// ---- Mian/MAIN.TcPOU
// Disclaimer
// 
// This publication contains statements about the suitability of our products for certain areas of application. These statements are based on typical features of our products. The examples shown in this publication are for demonstration purposes only. 
// The information provided herein should not be regarded as specific operation characteristics. It is incumbent on the customer to check and decide whether a product is suitable for use in a particular application. 
// We do not give any warranty that the source code which is made available with this publication is complete or accurate. 
//
// THE SAMPLE CODE CONTAINED IN THIS PUBLICATION IS PROVIDED “AS IS” WITHOUT WARRANTY OF ANY KIND, EITHER EXPRESSED, IMPLIED OR STATUTORY, INCLUDING WITHOUT LIMITATION, ANY WARRANTY WITH RESPECT TO NON-INFRINGEMENT, FREEDOM FROM PROPRIETARY RIGHTS OF THIRD PARTIES OR FITNESS FOR ANY PARTICULAR PURPOSE. 
// This publication may be changed from time to time without prior notice. No liability is assumed for errors and/or omissions. Our products are described in detail in our data sheets and documentations. Product-specific warnings and cautions must be observed. 
// For the latest version of our data sheets and documentations visit our website (www.beckhoff.de). 
//
// © Beckhoff Automation GmbH & Co. KG, 2022
// The reproduction, distribution and utilization of this document as well as the communication of its contents to others without express authorization is prohibited. Offenders will be held liable for the payment of damages. All rights reserved in the event of the grant of a patent, utility model or design.
PROGRAM MAIN
VAR_INPUT
	bExecuteComplete			: BOOL;									//Command Execute Complete, not defined
END_VAR
VAR
	firstCycle : BOOL := TRUE;
	UserModeCofig				: PML_UnitModeConfig;					//User can configure his own Mode
	
	fbMachine					: FB_Machine;							//Instance of FB_Machine
//	fbMachine_2					: FB_Machine;							//Instance of FB_Machine
	bMachineStartedUp			: BOOL := FALSE;						//TRUE, when first PLC-Cycle finish
	fbVisu						: FB_Visu;								//Visualization
							//Visualization
	fbTrigger					: F_TRIG;								//Trigger for resseting Counters
	fbTrigger_2					: F_TRIG;								//Trigger for resseting Counters

	fbLocalSystemTime			 : FB_LocalSystemTime;					//Get local Systemtime
	fbLocalSystemTime_2			 : FB_LocalSystemTime;					//Get local Systemtime
	
	fbTriggerErrorMainAxis		: R_TRIG;								//Trigger for detecting Error on Mainaxis and write into PackTags
	fbTriggerErrorMetalAxis		: R_TRIG;								//Trigger for detecting Error on Metalaxis and write into PackTags
	fbTriggerErrorPlasticAxis	: R_TRIG;								//Trigger for detecting Error on Plasticaxis and write into PackTags
	
	nStateCommandCheck			: DINT;									//State to handle with statecommands
	
	i	: INT;
	tonDly	: TON;
	FB_GetUPSStatus: FB_GetUPSStatus;	
	dataloaded: BOOL;								//UPS数据文件读取状态（True为读取成功，False为读取失败）
	OldData: BOOL;									//UPS备份数据文件读取状态
	PersistentDataStatus: EPlcPersistentStatus;		//Persistent数据读取（恢复）状态	
//	fb_ups	:FB_S_UPS_CX51x0;
	//application	: FB_Application;

	bButton				: BOOL;
	ton_button			: TON;

	refMachine_control_cmd	:REFERENCE TO MachineControlCommand;
	
	refMachine_control_cmd_2	:REFERENCE TO MachineControlCommand;
	
	rTrig_error	:ARRAY[0..10] OF R_TRIG;
	rTrig_error_2	:ARRAY[0..10] OF R_TRIG;
	
	rTrig_agingTest	:R_TRIG;
	fTrig_agingTest	:F_TRIG;

	topicCallbackTest	: E_Topics;
	dataCallbackTest	: PubSubData;
	topic_sample	: E_topic_sample;
	
	(***********************ADS********************************)
	light_tower_1			:	FB_Light_tower_module;
	light_tower_2			:	FB_Light_tower_module;
   // application_1			:	FB_Application;
	tote_1					:	FB_Tote_Subsystem;
	tote_2					:	FB_Tote_Subsystem;
	safety_1				:	FB_Safety_Subsystem;
	safety_2				:	FB_Safety_Subsystem;
	machine_control_1		:	FB_MachineControl_Subsystem;
	machine_control_2		:	FB_MachineControl_Subsystem;
	heartbeat_1				:	FB_HeartBeat_Subsystem;
	heartbeat_2				:	FB_HeartBeat_Subsystem;
	
	air_pressure_1			:	FB_AirPressure_Subsystem;
	air_pressure_2			:	FB_AirPressure_Subsystem;
	
	
	heartbeat_data_test : HeartbeatParams;	
	update_light_tower_params_test	: UpdateLightTowerParams;
	tset1: UDINT;
	
	
	version 				:	STRING(255);
	testbool: BOOL;
	inbound_tote_params_test : InboundToteParams;
	OutboundToteParams_test		:	OutboundToteParams;
	testbool1: BOOL;
	
	
	
	fbMachine1					: FB_Machine;							//Instance of FB_Machine
	fbMachine2					: FB_Machine;							//Instance of FB_Machine
	stateMachine1	: FB_StateMachine;
	stateMachine2	: FB_StateMachine;
	
	
END_VAR

(**************************************UPS*****************************************)
FB_GetUPSStatus(
	sNetId:= , 					//默认为本机Netid
	nPort:= , 					//ADS端口号，若不填写功能块会自动获取，默认0
	bEnable:= , 				//高电平有效，置True后循环读取UPS状态
	bValid=> , 					//当bValid为True时，stStatus的值有效
	bError=> , 
	nErrId=> , 
	stStatus=> );				//包含UPS信息的结构体
	

dataloaded:=_Appinfo.BootDataLoaded;
OldData:=_Appinfo.OldBootData;
PersistentDataStatus:=_Appinfo.PersistentStatus;

//application();
version:='v1.0.0';

tonDly(PT:= T#10MS);
//Configure Usermode 1
A_UnitModeConfig();

//Runs the first PLC-Cycle
IF fbMachine1.bUndefinedDone AND fbMachine2.bUndefinedDone AND NOT bMachineStartedUp THEN
	GVL.PackTags1.Command.CntrlCmd	:= ePMLCommand_Abort;
	GVL.PackTags2.Command.CntrlCmd	:= ePMLCommand_Abort;
	bMachineStartedUp			:= TRUE;
END_IF


GVL.bButtonProductionReq := GVL.PackTags.Command.UnitMode = ePMLProtUnitMode_Production AND GVL.PackTags.Status.UnitModeCurrent <> GVL.PackTags.Command.UnitMode;

//Set the Packtags
M_SetPackTags();

//set the errors and warnings in Packtags
M_SetPackTagsErrorWarning();

//Call Visu
M_CallVisu();
///////////////////initialize unitmode and set 
IF GVL.PackTags.Command.UnitMode=ePMLProtUnitMode_Invalid THEN
	GVL.PackTags.Command.UnitMode	:= ePMLProtUnitMode_Production;
	GVL.PackTags.Command.Parameter[1].Value := 1;
	GVL.PackTags1.Command.UnitMode	:= ePMLProtUnitMode_Production;
	GVL.PackTags1.Command.Parameter[1].Value := 1;	
	GVL.PackTags2.Command.UnitMode	:= ePMLProtUnitMode_Production;
	GVL.PackTags2.Command.Parameter[1].Value := 1;	
	
END_IF

//Call FB_Machine
GVL.fb_working1._iModuleID:= ModuleID.WORKING1;
GVL.fb_working1._sInstanceName	:= 'working1';
GVL.fb_loading._iModuleID:= ModuleID.LOADING;
GVL.fb_loading._sInstanceName	:= 'loading';
GVL.fb_working2._iModuleID:= ModuleID.WORKING2;
GVL.fb_working2._sInstanceName	:= 'working2';
GVL.fb_loading();
GVL.fb_working1();
GVL.fb_working2();
GVL.fb_autoStore1();
GVL.fb_autoStore1._sInstanceName	:= 'autoStore_1';
GVL.fb_autoStore1._iModuleID	:= ModuleID.AUTOSTORE1;
GVL.fb_autoStore2();
GVL.fb_autoStore2._sInstanceName	:= 'autoStore_2';
GVL.fb_autoStore2._iModuleID	:= ModuleID.AUTOSTORE2;

fbMachine1(	eModeCommand:= GVL.PackTags.Command.UnitMode,
  			eMode => GVL.PackTags1.Status.UnitModeCurrent, 
			eState =>GVL.PackTags1.Status.StateCurrent,
			pPML_Instance1:=ADR(GVL.fb_working1),
			pPML_Instance2:=ADR(GVL.fb_loading),
			pPackTags:=ADR(GVL.PackTags1),
			pSafetySystem	:= ADR(safety_1)
			);
			
fbMachine2(	eModeCommand:= GVL.PackTags.Command.UnitMode,
  			eMode => GVL.PackTags2.Status.UnitModeCurrent, 
			eState =>GVL.PackTags2.Status.StateCurrent,
			pPML_Instance1:=ADR(GVL.fb_working2),
			pPML_Instance2:=ADR(GVL.fb_loading),
			pPackTags:=ADR(GVL.PackTags2),
			pSafetySystem	:= ADR(safety_2)
			);		
	
stateMachine1(	pPackTags:=ADR(GVL.PackTags1),
				pMachine:=ADR(fbMachine1),
				pMachine_control_cmd := ADR(machine_control_1.machineControlCmd),
				pAirSystem	:=ADR(air_pressure_1),
				pSafetySystem	:= ADR(safety_1),
				pMcp	:= ADR(GVL.fb_mcp_1)
				);

stateMachine2(	pPackTags:=ADR(GVL.PackTags2),
				pMachine:=ADR(fbMachine2),
				pMachine_control_cmd := ADR(machine_control_2.machineControlCmd),
				pAirSystem	:=ADR(air_pressure_2),
				pSafetySystem	:= ADR(safety_2),
				pMcp	:= ADR(GVL.fb_mcp_2)
				);			
		
			
GVL.fbWriteLog(
	bWrite:= GVL.bWrite, 
	sFileName:= , 
	sMessage:= , 
	OK=> , 
	Busy=> , 
	ErrorMsg=> , 
	bError=> , 
	ErrorID=> );
	
(***********************ADS********************************)
GVL.fb_mcp_1(id:=1);
GVL.fb_mcp_2(id:=2);
tote_1();
safety_1(pHeartBeat:=ADR(heartbeat_1),pSafety_door:=ADR(GVL.fb_mcp_1.st_safety_door),pPackTags:=ADR(GVL.PackTags1),pMachine:=ADR(fbMachine1));
air_pressure_1(pPackTags:=ADR(GVL.PackTags1));
heartbeat_1();
light_tower_1(pHeartBeat:=ADR(heartbeat_1),pLightTower:= ADR(GVL.fb_mcp_1.lightTower));
machine_control_1(pMachineCurrentStatus:= ADR(GVL.PackTags1.Status.StateCurrent));
tote_1._sInstanceName	:='tote_1';
safety_1._sInstanceName	:='safety_1';
air_pressure_1._sInstanceName	:='air_pressure1';

tote_2();
light_tower_2(pHeartBeat:=ADR(heartbeat_2),pLightTower:= ADR(GVL.fb_mcp_2.lightTower));
safety_2(pHeartBeat:=ADR(heartbeat_2),pSafety_door:=ADR(GVL.fb_mcp_2.st_safety_door),pPackTags:=ADR(GVL.PackTags2),pMachine:=ADR(fbMachine2));
air_pressure_2(pPackTags:=ADR(GVL.PackTags2));
heartbeat_2();
machine_control_2(pMachineCurrentStatus:= ADR(GVL.PackTags2.Status.StateCurrent));
tote_2._sInstanceName	:='tote_2';
safety_2._sInstanceName	:='safety_2';
air_pressure_2._sInstanceName	:='air_pressure2';


M_SetUnitInfo();

ACTION A_UnitModeConfig:
UserModeCofig(
	eMode							:= ePMLUnitMode_Service, 
	bDisableClearing				:= TRUE, 
	bDisableStarting				:= FALSE, 
	bDisableSuspended				:= FALSE, 
	bDisableStopping				:= TRUE, 
	bDisableAborting				:= TRUE, 
	bDisableHolding					:= TRUE, 
	bDisableHeld					:= TRUE, 
	bDisableUnholding				:= TRUE, 
	bDisableSuspending				:= TRUE, 
	bDisableUnsuspending			:= TRUE, 
	bDisableResetting				:= TRUE, 
	bDisableIdle					:= FALSE, 
	bDisableCompleting				:= TRUE, 
	bDisableComplete				:= FALSE, 
	bEnableUnitModeChangeStopped	:= TRUE, 
	bEnableUnitModeChangeIdle		:= TRUE, 
	bEnableUnitModeChangeSuspended	:= FALSE, 
	bEnableUnitModeChangeExecute	:= FALSE, 
	bEnableUnitModeChangeAborted	:= TRUE, 
	bEnableUnitModeChangeHeld		:= FALSE, 
	bEnableUnitModeChangeComplete	:= TRUE, 
	bError							=> , 
	nErrorId						=> );
UserModeCofig(
	eMode							:= ePMLUnitMode_Production, 
	bDisableClearing				:= FALSE, 
	bDisableStarting				:= FALSE, 
	bDisableSuspended				:= TRUE, 
	bDisableStopping				:= FALSE, 
	bDisableAborting				:= FALSE, 
	bDisableHolding					:= TRUE, 
	bDisableHeld					:= TRUE, 
	bDisableUnholding				:= TRUE, 
	bDisableSuspending				:= TRUE, 
	bDisableUnsuspending			:= TRUE, 
	bDisableResetting				:= FALSE, 
	bDisableIdle					:= FALSE, 
	bDisableCompleting				:= FALSE, 
	bDisableComplete				:= FALSE, 
	bEnableUnitModeChangeStopped	:= TRUE, 
	bEnableUnitModeChangeIdle		:= TRUE, 
	bEnableUnitModeChangeSuspended	:= FALSE, 
	bEnableUnitModeChangeExecute	:= FALSE, 
	bEnableUnitModeChangeAborted	:= TRUE, 
	bEnableUnitModeChangeHeld		:= FALSE, 
	bEnableUnitModeChangeComplete	:= TRUE, 
	bError							=> , 
	nErrorId						=> );
END_ACTION

METHOD M_CallVisu
VAR_INPUT
END_VAR
//Calling FB_Visu
fbVisu(
	aKeyPressed				:= GVL.aKeyPressed,
	aUnitInfo				:= GVL.aUnitInfo, 
	bInvalidEntry			=> ,
	aCaption				=> GVL.aCaption,
	eModeVisu				=> ,
	eStateVisu				=> ,
	sUnitName				=> ,
	iFrameVisible			=> );
END_METHOD

METHOD M_SetPackTags
VAR_INPUT
END_VAR
VAR	
END_VAR
//***************************Writing Data into GVL.PackTags***************************

//Parameters for the production
GVL.PackTags.Command.Parameter[1].ID				:= 1;
GVL.PackTags.Command.Parameter[1].Name				:= 'Quantity';
GVL.PackTags.Command.Parameter[1].Unit				:= 'Tote';

//Countig produced totes, see fb_sample1
GVL.PackTags.Admin.ProdProcessedCount[1].ID			:= 1;
GVL.PackTags.Admin.ProdProcessedCount[1].Name		:= 'ToteFinish_Sample';
GVL.PackTags.Admin.ProdProcessedCount[1].Unit		:= 'Tote';





//Write the actual state and mode into the GVL.PackTags
GVL.PackTags.Status.StateCurrent					:= fbMachine1.eState;
GVL.PackTags.Status.UnitModeCurrent					:= fbMachine1.eMode;
GVL.PackTags.Status.StateRequested					:= fbMachine1.eCommand;
GVL.PackTags.Status.UnitModeRequested				:= fbMachine1.eModeCommand;
GVL.PackTags.Status.StateChangeInProcess			:= GVL.PackTags.Status.StateCurrent <> GVL.PackTags.Status.StateRequested;
GVL.PackTags.Status.UnitModeChangeInProcess			:= GVL.PackTags.Status.UnitModeCurrent <> GVL.PackTags.Status.UnitModeRequested;

//Write the actual state and mode into the GVL.PackTags2
GVL.PackTags1.Status.StateCurrent					:= fbMachine1.eState;
GVL.PackTags1.Status.UnitModeCurrent					:= fbMachine1.eMode;
GVL.PackTags1.Status.StateRequested					:= fbMachine1.eCommand;
GVL.PackTags1.Status.UnitModeRequested				:= fbMachine1.eModeCommand;
GVL.PackTags1.Status.StateChangeInProcess			:= GVL.PackTags1.Status.StateCurrent <> GVL.PackTags1.Status.StateRequested;
GVL.PackTags1.Status.UnitModeChangeInProcess			:= GVL.PackTags1.Status.UnitModeCurrent <> GVL.PackTags1.Status.UnitModeRequested;
//Write the actual state and mode into the GVL.PackTags2
GVL.PackTags2.Status.StateCurrent					:= fbMachine2.eState;
GVL.PackTags2.Status.UnitModeCurrent					:= fbMachine2.eMode;
GVL.PackTags2.Status.StateRequested					:= fbMachine2.eCommand;
GVL.PackTags2.Status.UnitModeRequested				:= fbMachine2.eModeCommand;
GVL.PackTags2.Status.StateChangeInProcess			:= GVL.PackTags2.Status.StateCurrent <> GVL.PackTags2.Status.StateRequested;
GVL.PackTags2.Status.UnitModeChangeInProcess			:= GVL.PackTags2.Status.UnitModeCurrent <> GVL.PackTags2.Status.UnitModeRequested;


//Write actual time and date in GVL.PackTags
fbLocalSystemTime(sNetID:= '', bEnable := TRUE);
GVL.PackTags.Admin.PlcDateTime[0]	:= fbLocalSystemTime.systemTime.wYear;
GVL.PackTags.Admin.PlcDateTime[1]	:= fbLocalSystemTime.systemTime.wMonth;
GVL.PackTags.Admin.PlcDateTime[2]	:= fbLocalSystemTime.systemTime.wDay;
GVL.PackTags.Admin.PlcDateTime[3]	:= fbLocalSystemTime.systemTime.wHour;
GVL.PackTags.Admin.PlcDateTime[4]	:= fbLocalSystemTime.systemTime.wMinute;
GVL.PackTags.Admin.PlcDateTime[5]	:= fbLocalSystemTime.systemTime.wSecond;
GVL.PackTags.Admin.PlcDateTime[6]	:= fbLocalSystemTime.systemTime.wMilliseconds;
GVL.PackTags1.Admin.PlcDateTime	:= GVL.PackTags.Admin.PlcDateTime;
GVL.PackTags2.Admin.PlcDateTime	:= GVL.PackTags.Admin.PlcDateTime;
//Set the productcounter to 0, when the production command is completed
fbTrigger(CLK:= (fbMachine1.eState = ePMLState_Complete));
IF fbTrigger.Q OR GVL.stChangeIntoProduction.bYesReset THEN
	GVL.PackTags1.Admin.ProdProcessedCount[1].Count	:= 0;
	GVL.PackTags1.Command.Parameter[1].Value			:= 0;
	GVL.nVisuProductCommand							:= 0;
END_IF

//Set the productcounter to 0, when the production command is completed
fbTrigger(CLK:= (fbMachine2.eState = ePMLState_Complete));
IF fbTrigger.Q OR GVL.stChangeIntoProduction.bYesReset THEN
	GVL.PackTags2.Admin.ProdProcessedCount[1].Count	:= 0;
	GVL.PackTags2.Command.Parameter[1].Value			:= 0;
	GVL.nVisuProductCommand							:= 0;
END_IF
END_METHOD

METHOD M_SetPackTagsErrorWarning
VAR_INPUT
END_VAR
//====================Error and Warnig setting========================
//Warnings
GVL.PackTags1.Admin.Warning[1].Message	:= 'Invalid Production Command, command Products must be higher than 0';
GVL.PackTags1.Admin.Warning[1].ID 		:= 1;

GVL.PackTags1.Admin.Warning[2].Message	:= 'Invalid Mode Command, please try anothereone';
GVL.PackTags1.Admin.Warning[2].ID		:= 2;


//====================Error and Warnig handling========================
//warning for invalid production command
IF 	GVL.PackTags1.Status.UnitModeCurrent = ePMLProtUnitMode_Production AND 
	GVL.PackTags1.Status.StateCurrent = ePMLState_Idle AND 
	GVL.PackTags1.Command.CntrlCmd = ePMLCommand_Start AND
 	GVL.PackTags1.Command.Parameter[1].Value <= 0 
THEN
	GVL.PackTags1.Admin.Warning[1].Trigger :=TRUE;
ELSE
	GVL.PackTags1.Admin.Warning[1].Trigger :=FALSE;
END_IF

//warning for invalid mode command
IF fbMachine1.bInvalidModeCommandOut THEN
	GVL.PackTags1.Admin.Warning[2].Trigger :=TRUE;
ELSE 
	GVL.PackTags1.Admin.Warning[2].Trigger :=FALSE;
END_IF





//====================Error and Warnig setting========================
//Warnings
GVL.PackTags1.Admin.Warning[1].Message	:= 'Invalid Production Command, command Products must be higher than 0';
GVL.PackTags1.Admin.Warning[1].ID 		:= 1;

GVL.PackTags1.Admin.Warning[2].Message	:= 'Invalid Mode Command, please try anothereone';
GVL.PackTags1.Admin.Warning[2].ID		:= 2;


//====================Error and Warnig handling========================
//warning for invalid production command
IF 	GVL.PackTags2.Status.UnitModeCurrent = ePMLProtUnitMode_Production AND 
	GVL.PackTags2.Status.StateCurrent = ePMLState_Idle AND 
	GVL.PackTags2.Command.CntrlCmd = ePMLCommand_Start AND
 	GVL.PackTags2.Command.Parameter[1].Value <= 0 
THEN
	GVL.PackTags2.Admin.Warning[1].Trigger :=TRUE;
ELSE
	GVL.PackTags2.Admin.Warning[1].Trigger :=FALSE;
END_IF

//warning for invalid mode command
IF fbMachine2.bInvalidModeCommandOut THEN
	GVL.PackTags2.Admin.Warning[2].Trigger :=TRUE;
ELSE 
	GVL.PackTags2.Admin.Warning[2].Trigger :=FALSE;
END_IF
END_METHOD

METHOD M_SetUnitInfo
VAR_INPUT
END_VAR
GVL.aUnitInfo[eMachine1].Name			:= 'fbMachine1';
GVL.aUnitInfo[eMachine1].ActMode			:= fbMachine1.eMode;
GVL.aUnitInfo[eMachine1].ActState		:= fbMachine1.eState;

GVL.aUnitInfo[eMachine1].Name			:= 'fbMachine2';
GVL.aUnitInfo[eMachine1].ActMode		:= fbMachine2.eMode;
GVL.aUnitInfo[eMachine1].ActState		:= fbMachine2.eState;

//GVL.aUnitInfo[eSample].Name				:= GVL.fb_sample._sInstanceName;
//GVL.aUnitInfo[eSample].ActMode			:= GVL.fb_sample.eMode;
//GVL.aUnitInfo[eSample].ActState			:= GVL.fb_sample.eState;


GVL.aUnitInfo[eLoading].Name			:= GVL.fb_loading._sInstanceName;
GVL.aUnitInfo[eLoading].ActMode			:= GVL.fb_loading.eMode;
GVL.aUnitInfo[eLoading].ActState		:= GVL.fb_loading.eState;


GVL.aUnitInfo[eWorking1].Name			:= GVL.fb_working1._sInstanceName;
GVL.aUnitInfo[eWorking1].ActMode		:= GVL.fb_working1.eMode;
GVL.aUnitInfo[eWorking1].ActState		:= GVL.fb_working1.eState;


GVL.aUnitInfo[eWorking2].Name			:= GVL.fb_working2._sInstanceName;
GVL.aUnitInfo[eWorking2].ActMode		:= GVL.fb_working2.eMode;
GVL.aUnitInfo[eWorking2].ActState		:= GVL.fb_working2.eState;
END_METHOD

END_PROGRAM

// ---- Mian/FB_StateMachine.TcPOU
FUNCTION_BLOCK FB_StateMachine
VAR_INPUT
	
	pPackTags				: POINTER TO ST_PackMLv30;
	pMachine				: POINTER TO FB_Machine;	
	pMachine_control_cmd	: POINTER TO MachineCommandStructure;	
	pAirSystem				: POINTER TO FB_AirPressure_Subsystem;
	pSafetySystem			: POINTER TO FB_Safety_Subsystem;	
	pMcp					: POINTER TO FB_mcp;
END_VAR
VAR_OUTPUT
END_VAR
VAR
	rTrig_error	:ARRAY[1..10] OF R_TRIG;
	i	: INT;
		

END_VAR

(*command from 1:PLC HMI buttons;2:APP;3:Safety module;4:each modules*)
/////////////////////////////abort/////////////////////////////	
IF 	pMachine^.eState <> ePMLState_Aborted AND pMachine^.eState <> ePMLState_Clearing THEN	
	IF pPackTags^.Command.CntrlCmd = ePMLCommand_Abort OR M_CheckError() THEN
		IF pMachine^.M_UnitsActive(ePMLCommand_Abort) THEN
			pMachine^.eCommand	:= ePMLCommand_Abort;
			pMachine_control_cmd^.command	:= MachineControlCommand.DO_NOTHING;
		END_IF
	END_IF
END_IF
/////////////////////////////stop/////////////////////////////
IF M_CheckError() THEN
	//
ELSE					
	IF (pPackTags^.Command.CntrlCmd = ePMLCommand_Stop OR 
		pMachine_control_cmd^.command = MachineControlCommand.STOP OR 
		pSafetySystem^.pml_command=ePMLCommand_Stop) AND pMachine^.eState <> ePMLState_Stopped
	THEN
		IF pMachine^.M_UnitsActive(ePMLCommand_Stop) THEN
			pMachine^.eCommand	:= ePMLCommand_Stop;
		END_IF
	END_IF
END_IF

CASE pMachine^.eState OF
			
	ePMLState_Aborted:
		IF pMcp^.st_safety_door.button_reset THEN
			pPackTags^.Command.CntrlCmd := ePMLCommand_Clear;
		END_IF
		IF 	pPackTags^.Command.CntrlCmd = ePMLCommand_Clear OR
			(pSafetySystem^.safety_status=SafetyStatus.READY AND pMachine_control_cmd^.command=MachineControlCommand.RESET)//while safety is ready,can be reset remotely	 
		THEN
			IF pSafetySystem^.M_reset() THEN	//reset safety first
				IF pSafetySystem^.xError THEN
					pPackTags^.Command.CntrlCmd		:= ePMLCommand_Undefined;
					pMachine_control_cmd^.command	:= MachineControlCommand.DO_NOTHING;
				ELSE
					IF pMachine^.M_UnitsActive(ePMLCommand_Clear) THEN
						pMachine^.eCommand	:= ePMLCommand_Clear;
					END_IF					
				END_IF
			END_IF	
		END_IF
		//reset command
		IF pMachine^.eCommand = ePMLCommand_Abort THEN
			pMachine^.eCommand	:= ePMLCommand_Undefined;
		END_IF
			
	ePMLState_Complete:		
		IF (pPackTags^.Command.CntrlCmd = ePMLCommand_Reset OR pMachine_control_cmd^.command = MachineControlCommand.RESET (*OR
		 	pMcp^.st_safety_door.button_reset*)) 
		THEN
			pMachine^.eCommand	:= ePMLCommand_Reset;
		END_IF
			
			
	ePMLState_Idle:
		IF (pPackTags^.Command.CntrlCmd = ePMLCommand_Start OR pMachine_control_cmd^.command = MachineControlCommand.START)	AND
			(NOT (pPackTags^.Command.Parameter[1].Value <= 0) OR NOT (pMachine^.eMode = 1))
		THEN	
			IF pMachine^.M_UnitsActive(ePMLCommand_Start) THEN
				pMachine^.eCommand	:= ePMLCommand_Start;
			END_IF
		END_IF
		IF pMachine_control_cmd^.command = MachineControlCommand.RESET THEN
			pMachine_control_cmd^.command	:= MachineControlCommand.DO_NOTHING;
		END_IF
		//reset command
		IF pMachine^.eCommand = ePMLCommand_Reset THEN
			pMachine^.eCommand	:= ePMLCommand_Undefined;
		END_IF
			
			
	ePMLState_Stopped:
		IF pPackTags^.Command.CntrlCmd = ePMLCommand_Reset OR pMachine_control_cmd^.command = MachineControlCommand.RESET THEN		
			IF pMachine^.M_UnitsActive(ePMLCommand_Reset) THEN
				pMachine^.eCommand	:= ePMLCommand_Reset;
			END_IF
		END_IF		
		IF (pPackTags^.Command.CntrlCmd = ePMLCommand_Start OR pMachine_control_cmd^.command = MachineControlCommand.START)	AND
			(NOT (pPackTags^.Command.Parameter[1].Value <= 0) OR NOT (pMachine^.eMode = 1)) AND
			stPMLUnitModeConfiguration[pMachine^.eMode].aStateDisabled[ePMLState_Idle] 
		THEN	
			IF pMachine^.M_UnitsActive(ePMLCommand_Start) THEN
				pMachine^.eCommand	:= ePMLCommand_Start; 	
			END_IF			
		END_IF	
		IF pMachine_control_cmd^.command = MachineControlCommand.STOP THEN
			pMachine_control_cmd^.command	:= MachineControlCommand.DO_NOTHING;
		END_IF	
		//reset command
		IF pMachine^.eCommand = ePMLCommand_Clear OR pMachine^.eCommand = ePMLCommand_Stop THEN
			pMachine^.eCommand	:= ePMLCommand_Undefined;
		END_IF
			
			
	ePMLState_Execute:	
		IF pMachine_control_cmd^.command = MachineControlCommand.START THEN
			pMachine_control_cmd^.command	:= MachineControlCommand.DO_NOTHING;
		END_IF
		IF pPackTags^.Command.CntrlCmd = ePMLCommand_Hold	AND	
			(pMachine^.eMode =  1 OR pMachine^.eMode =  4 OR pMachine^.eMode = 2)  
		THEN
			pMachine^.eCommand	:= ePMLCommand_Hold;
		END_IF	
		IF pPackTags^.Command.CntrlCmd = ePMLCommand_Suspend AND (pMachine^.eMode = 4 OR pMachine^.eMode = 1)THEN
		 
			pMachine^.eCommand	:= ePMLCommand_Suspend;
		END_IF	 
		//reset command
		IF pMachine^.eCommand = ePMLCommand_Start THEN
			pMachine^.eCommand	:= ePMLCommand_Undefined;
		END_IF
			
			
	ePMLState_Held:	 
		IF pPackTags^.Command.CntrlCmd = ePMLCommand_Unhold THEN
			pMachine^.eCommand	:= ePMLCommand_Unhold;
		END_IF
			
			
	ePMLState_Suspended:
		IF pPackTags^.Command.CntrlCmd = ePMLCommand_Unsuspend THEN
			pMachine^.eCommand	:= ePMLCommand_Unsuspend;
		END_IF
			
			
	ePMLState_Aborting,ePMLState_Clearing,ePMLState_Resetting,ePMLState_Starting,ePMLState_Stopping:
		pPackTags^.Command.CntrlCmd	:= ePMLCommand_Undefined;

		
		
END_CASE

METHOD M_CheckError : BOOL

VAR
	
END_VAR
M_CheckError	:= FALSE;

FOR i:=1 TO GlobalParameters.MaxAlarms DO
	IF pPackTags^.Admin.Alarm[i].Trigger THEN
		M_CheckError	:= TRUE;
	END_IF
END_FOR
//RETURN;//remove this while safety and air is ready
IF pSafetySystem^.xError OR pAirSystem^.air_pressure_status=AirPressureStatus.ERROR THEN
	M_CheckError	:= TRUE;
END_IF
END_METHOD

END_FUNCTION_BLOCK

// ---- GlobalTextList.TcGTLO
TEXTLIST GlobalTextList
  1242 = '    UNKNOWN := 0 \n   VACANT :=  1\n      LOADED := 2\n AWAITING_INBOUND_AVAILABILITY := 3 \n      INBOUNDING := 4\n  AWAITING_OUTBOUND_AVAILABILITY:5\n    OUTBOUNDING := 6\n    PERTURBING := 7\n    UNKNOWN_ERROR := 50, \n    MECHANICAL_ERROR := 51,\n    ELECTRICAL_ERROR := 52,\n    SAFETY_ERROR := 53,\n    UPSTREAM_NOT_READY := 54,\n    TIMEOUT_WAITING_FOR_NEW_TOTE := 55,\n    DOWNSTREAM_NOT_READY := 56,\n    TIMEOUT_WAITING_FOR_SPACE := 57,\n\tBAG_OPEN_FAILED := 100'
  1602 = '    UNKNOWN := 0 \n   VACANT :=  1\n      LOADED := 2\n AWAITING_INBOUND_AVAILABILITY := 3, \n      INBOUNDING := 4,\n  AWAITING_OUTBOUND_AVAILABILITY:5, \n    OUTBOUNDING := 6,  \n    PERTURBING := 7, \n    UNKNOWN_ERROR := 50, \n    MECHANICAL_ERROR := 51,\n    ELECTRICAL_ERROR := 52,\n    SAFETY_ERROR := 53,\n    UPSTREAM_NOT_READY := 54,\n    TIMEOUT_WAITING_FOR_NEW_TOTE := 55,\n    DOWNSTREAM_NOT_READY := 56,\n    TIMEOUT_WAITING_FOR_SPACE := 57,\n\tBAG_OPEN_FAILED := 100'
  133 = '    UNKNOWN := 0 \n   VACANT :=  1\n      LOADED := 2 AWAITING_INBOUND_AVAILABILITY := 3, \n      INBOUNDING := 4,  AWAITING_OUTBOUND_AVAILABILITY:5, \n    OUTBOUNDING := 6,  \n    PERTURBING := 7, \n    UNKNOWN_ERROR := 50, \n    MECHANICAL_ERROR := 51,\n    ELECTRICAL_ERROR := 52,\n    SAFETY_ERROR := 53,\n    UPSTREAM_NOT_READY := 54,\n    TIMEOUT_WAITING_FOR_NEW_TOTE := 55,\n    DOWNSTREAM_NOT_READY := 56,\n    TIMEOUT_WAITING_FOR_SPACE := 57,\n\tBAG_OPEN_FAILED := 100'
  1738 = '    UNKNOWN := 0 \n   VACANT :=  1，\n      LOADED := 2，\n AWAITING_INBOUND_AVAILABILITY := 3, \n      INBOUNDING := 4,\n  AWAITING_OUTBOUND_AVAILABILITY:5, \n    OUTBOUNDING := 6,  \n    PERTURBING := 7, \n    UNKNOWN_ERROR := 50, \n    MECHANICAL_ERROR := 51,\n    ELECTRICAL_ERROR := 52,\n    SAFETY_ERROR := 53,\n    UPSTREAM_NOT_READY := 54,\n    TIMEOUT_WAITING_FOR_NEW_TOTE := 55,\n    DOWNSTREAM_NOT_READY := 56,\n    TIMEOUT_WAITING_FOR_SPACE := 57,\n\tBAG_OPEN_FAILED := 100'
  3042 = '    UNKNOWN := 0 \n   VACANT :=  1，\n      LOADED := 2，\n AWAITING_INBOUND_AVAILABILITY := 3, \n      INBOUNDING := 4,  AWAITING_OUTBOUND_AVAILABILITY:5, \n    OUTBOUNDING := 6,  \n    PERTURBING := 7, \n    UNKNOWN_ERROR := 50, \n    MECHANICAL_ERROR := 51,\n    ELECTRICAL_ERROR := 52,\n    SAFETY_ERROR := 53,\n    UPSTREAM_NOT_READY := 54,\n    TIMEOUT_WAITING_FOR_NEW_TOTE := 55,\n    DOWNSTREAM_NOT_READY := 56,\n    TIMEOUT_WAITING_FOR_SPACE := 57,\n\tBAG_OPEN_FAILED := 100'
  298 = '    UNKNOWN := 0 \n   VACANT :=  1，\n      LOADED := 2， AWAITING_INBOUND_AVAILABILITY := 3, \n      INBOUNDING := 4,  AWAITING_OUTBOUND_AVAILABILITY:5, \n    OUTBOUNDING := 6,  \n    PERTURBING := 7, \n    UNKNOWN_ERROR := 50, \n    MECHANICAL_ERROR := 51,\n    ELECTRICAL_ERROR := 52,\n    SAFETY_ERROR := 53,\n    UPSTREAM_NOT_READY := 54,\n    TIMEOUT_WAITING_FOR_NEW_TOTE := 55,\n    DOWNSTREAM_NOT_READY := 56,\n    TIMEOUT_WAITING_FOR_SPACE := 57,\n\tBAG_OPEN_FAILED := 100'
  387 = '    UNKNOWN := 0, \n    VACANT := 1\n    LOADED := 2,  AWAITING_INBOUND_AVAILABILITY := 3,  \n     INBOUNDING := 4,      AWAITING_OUTBOUND_AVAILABILITY := 5,  \n    OUTBOUNDING := 6,\n    PERTURBING := 7, \n    UNKNOWN_ERROR := 50, \n    MECHANICAL_ERROR := 51,\n    ELECTRICAL_ERROR := 52,\n    SAFETY_ERROR := 53,\n    UPSTREAM_NOT_READY := 54,\n    TIMEOUT_WAITING_FOR_NEW_TOTE := 55,\n    DOWNSTREAM_NOT_READY := 56,\n    TIMEOUT_WAITING_FOR_SPACE := 57,\n\t\n\tBAG_OPEN_FAILED := 100'
  1866 = '    UNKNOWN := 0, \n   VACANT :=  1,  \n      LOADED :=  2,  AWAITING_INBOUND_AVAILABILITY := 3, \n      INBOUNDING := 4,  AWAITING_OUTBOUND_AVAILABILITY:5, \n    OUTBOUNDING := 6,  \n    PERTURBING := 7, \n    UNKNOWN_ERROR := 50, \n    MECHANICAL_ERROR := 51,\n    ELECTRICAL_ERROR := 52,\n    SAFETY_ERROR := 53,\n    UPSTREAM_NOT_READY := 54,\n    TIMEOUT_WAITING_FOR_NEW_TOTE := 55,\n    DOWNSTREAM_NOT_READY := 56,\n    TIMEOUT_WAITING_FOR_SPACE := 57,\n\tBAG_OPEN_FAILED := 100'
  2213 = '    UNKNOWN := 0, \n   VACANT := 1,  \n    LOADED := 2,  AWAITING_INBOUND_AVAILABILITY := 3, \n      INBOUNDING := 4,  AWAITING_OUTBOUND_AVAILABILITY:5, \n    OUTBOUNDING := 6,  \n    PERTURBING := 7, \n    UNKNOWN_ERROR := 50, \n    MECHANICAL_ERROR := 51,\n    ELECTRICAL_ERROR := 52,\n    SAFETY_ERROR := 53,\n    UPSTREAM_NOT_READY := 54,\n    TIMEOUT_WAITING_FOR_NEW_TOTE := 55,\n    DOWNSTREAM_NOT_READY := 56,\n    TIMEOUT_WAITING_FOR_SPACE := 57,\n\tBAG_OPEN_FAILED := 100'
  972 = '    UNKNOWN := 0, \n   VACANT := 1,  \n    LOADED := 2,  AWAITING_INBOUND_AVAILABILITY := 3,  \n      INBOUNDING := 4,  AWAITING_OUTBOUND_AVAILABILITY := 5,  \n    OUTBOUNDING := 6,  \n    PERTURBING := 7, \n    UNKNOWN_ERROR := 50, \n    MECHANICAL_ERROR := 51,\n    ELECTRICAL_ERROR := 52,\n    SAFETY_ERROR := 53,\n    UPSTREAM_NOT_READY := 54,\n    TIMEOUT_WAITING_FOR_NEW_TOTE := 55,\n    DOWNSTREAM_NOT_READY := 56,\n    TIMEOUT_WAITING_FOR_SPACE := 57,\n\t\n\tBAG_OPEN_FAILED := 100'
  599 = '    UNKNOWN := 0, \n   VACANT := 1,  \n    LOADED := 2,  AWAITING_INBOUND_AVAILABILITY := 3,  \n      INBOUNDING := 4,  AWAITING_OUTBOUND_AVAILABILITY := 5,  \n    OUTBOUNDING := 6,  \n    PERTURBING := 7, \n    UNKNOWN_ERROR := 50, \n    MECHANICAL_ERROR := 51,\n    ELECTRICAL_ERROR := 52,\n    SAFETY_ERROR := 53,\n    UPSTREAM_NOT_READY := 54,\n    TIMEOUT_WAITING_FOR_NEW_TOTE := 55,\n    DOWNSTREAM_NOT_READY := 56,\n    TIMEOUT_WAITING_FOR_SPACE := 57,\n\tBAG_OPEN_FAILED := 100'
  2173 = '    UNKNOWN := 0,  (* when system is down *)\n    VACANT := 1, (* no tote here *)\n    LOADED := 2,  (* a tote loaded in current position *)\n    AWAITING_INBOUND_AVAILABILITY := 3,  (* waiting for an available inbound tote *)\n    INBOUNDING := 4,  (* inbounding tote from upper line *)\n    AWAITING_OUTBOUND_AVAILABILITY := 5,  (* waiting for an available outbound space *)\n    OUTBOUNDING := 6,  (* outbound tote to lower line *)\n    PERTURBING := 7, (* Tote vibrating *)\n\n    UNKNOWN_ERROR := 50, (* in error state, we should extend the error in the future\t*)\n    MECHANICAL_ERROR := 51,\n    ELECTRICAL_ERROR := 52,\n    SAFETY_ERROR := 53,\n    UPSTREAM_NOT_READY := 54,\n    TIMEOUT_WAITING_FOR_NEW_TOTE := 55,\n    DOWNSTREAM_NOT_READY := 56,\n    TIMEOUT_WAITING_FOR_SPACE := 57,\n\t\n\tBAG_OPEN_FAILED := 100'
  55 = ' command Products: %i'
  323 = '%.2f'
  206 = '%.2f mm'
  829 = '%.2f MPa'
  1131 = '%.2r'
  740 = '%.3f mm'
  201 = '%s'
  209 = '+'
  210 = '-'
  2384 = '2 Systems'
  54 = 'A C C I D E N T'
  18 = 'Abort'
  394 = 'ABORT INBOUND'
  2668 = 'ABORT OUTBOUND'
  33 = 'Aborted'
  34 = 'Aborting'
  602 = 'Acc'
  843 = 'Actual Position'
  830 = 'Admin'
  773 = 'Aging test'
  5 = 'Alarm'
  61 = 'Average MachSpeed: %5.2f Package/min'
  203 = 'Axis Error '
  299 = 'Axis_bagOpen_0'
  618 = 'Axis_bagOpen_1'
  211 = 'Axis_bagOpen_2'
  743 = 'Axis_bagOpen_3'
  324 = 'Axis_vacuun_0'
  786 = 'Axis_vacuun_1'
  317 = 'BAFFLE SENSOR1'
  1963 = 'BAFFLE SENSOR2'
  179 = 'BagOpen'
  63 = 'BagOpening'
  11 = 'BagOpening '
  521 = 'BagOpening-1'
  1064 = 'BagOpening_1'
  2321 = 'BagOpening_2'
  2069 = 'BagOpening_Detection'
  959 = 'Bag_)'
  1353 = 'Bag_0'
  1316 = 'Bag_1'
  1317 = 'Bag_closed'
  517 = 'Bag_opened'
  1009 = 'Bag_preopen'
  2196 = 'bDisplay'
  81 = 'BELT ESTOP'
  1803 = 'bLoad_up'
  808 = 'Breaker OFF'
  486 = 'Breaker ON'
  2216 = 'Btton Start'
  1159 = 'buffer'
  327 = 'BUFFER SAFETY'
  732 = 'Buffer Stopper'
  481 = 'bUsingOpenBag'
  1712 = 'Button stop'
  1438 = 'b_EStopRestart'
  16 = 'Clear'
  32 = 'Clearing'
  17 = 'Command'
  38 = 'Complete'
  1085 = 'Completing'
  58 = 'CurrentMachSpeed:%5.2f Package/min'
  1975 = 'DateTime'
  1723 = 'Datetime'
  349 = 'Dec'
  216 = 'deg/s'
  217 = 'deg/s²'
  50 = 'Detection\nof metal'
  180 = 'DIO'
  68 = 'Do you want to change tp production mode?'
  662 = 'DOG'
  2636 = 'DOOR CLOSED'
  2225 = 'Door Closed'
  1080 = 'Down'
  673 = 'error'
  586 = 'EStop Restart'
  2274 = 'EStopRestart'
  23 = 'Execute'
  19 = 'Execute\nComplete'
  924 = 'Extend'
  2482 = 'extend'
  614 = 'extended'
  59 = 'Finished Metalboxes: %i'
  60 = 'Finished Plasticboxes: %i'
  56 = 'Finished Products: %i '
  801 = 'Flood Light'
  1197 = 'GVL_IOLink'
  25 = 'Held'
  12 = 'Hold'
  26 = 'Holding'
  841 = 'HOME'
  248 = 'HomeDone'
  902 = 'ID'
  21 = 'Idle'
  136 = 'inbound'
  134 = 'INBOUND'
  710 = 'inbound_1'
  1624 = 'inbound_2'
  44 = 'INIT'
  4 = 'Invalid'
  1037 = 'Lamp'
  2490 = 'LIFT DOOR LEFT'
  2284 = 'LIFT DOOR RIGHT'
  668 = 'LIFT STO EDM'
  473 = 'Lift_down'
  293 = 'Lift_iuo'
  316 = 'Lift_up'
  51 = 'Light\nsensor'
  2749 = 'LIGHT STO EDM'
  319 = 'Load'
  1648 = 'Load Tote'
  1129 = 'Load Tote Request'
  762 = 'Loading'
  416 = 'Load_up'
  581 = 'Lock MCP Left Door'
  222 = 'Lock MCP Right Door'
  580 = 'Log In'
  234 = 'Log Out'
  1496 = 'LogOut'
  6 = 'Mantainance'
  7 = 'Manual'
  2290 = 'MCP ESTOP LEFT'
  1000 = 'MCP ESTOP RIGHT'
  1593 = 'MCP ESTOP2'
  708 = 'Message'
  361 = 'Method'
  2239 = 'MID SAFETY DOOR1'
  2485 = 'MID SAFETY DOOR2'
  52 = 'Move belt\n+'
  53 = 'Move to\nwork position'
  491 = 'Muanal'
  737 = 'name'
  3 = 'No'
  1516 = 'NO.'
  258 = 'NO. '
  1043 = 'None'
  1736 = 'Open MCP Left Door'
  1323 = 'Open MCP Right Door'
  711 = 'Operator'
  1406 = 'OUTBOUND'
  381 = 'outbound_1'
  1368 = 'outbound_2'
  1318 = 'outbound_assist\n\n'
  760 = 'outbound_assist_1\n\n'
  182 = 'outbound_assist_2\n\n'
  1029 = 'outbound_end'
  787 = 'Pause'
  1446 = 'photosensor'
  2037 = 'photo_sensor_bottom'
  1081 = 'photo_sensor_diagonal'
  706 = 'photo_sens[1]or_start'
  1231 = 'PICKMODULE STO EDM'
  882 = 'PICKMODULE2 STO EDM'
  1922 = 'PLACE1 STO EDM'
  1263 = 'PLACE2 STO EDM'
  1450 = 'PML '
  598 = 'Position Setting'
  1051 = 'Production'
  57 = 'Reset the Visu'
  30 = 'Reseting'
  176 = 'ROBO2T ESTOP'
  40 = 'ROBOT1 EAS'
  1399 = 'ROBOT1 EES'
  2581 = 'ROBOT1 ESTOP'
  1167 = 'ROBOT2 EAS'
  2067 = 'ROBOT2 EES'
  1126 = 'ROLLER BELT STO EDM'
  1023 = 'rolleroutbound_assist\n\n'
  1305 = 'roller_assign'
  1160 = 'roller_inbound'
  1610 = 'roller_inbound_assist'
  2157 = 'roller_outbound'
  1295 = 'roller_outbound_assist\n\n'
  2362 = 'SAFETY DOOR LEFT'
  1331 = 'SAFETYDOOR RIGHT'
  1925 = 'Sample'
  36 = 'SC'
  1012 = 'sensor[0]'
  1257 = 'sensor[1]'
  82 = 'sensor[2]'
  774 = 'sensor[3]'
  1262 = 'sensor[4]'
  1137 = 'sensor[5]'
  794 = 'sensor[6]'
  512 = 'sensor[7]'
  2929 = 'sensor_lift_atDownPos'
  681 = 'sensor_start[0]'
  1006 = 'sensor_start[1]'
  2179 = 'sensor_transfer_atFeedingPos'
  3056 = 'sensor_transfer_atWorkingPos'
  62 = 'Seperated Boxes: %i'
  415 = 'Service'
  102 = 'sStepID'
  99 = 'Jerk'
  839 = 'JOG BW'
  840 = 'JOG FW'
  1374 = 'lift'
  795 = 'LIFT'
  178 = 'Lift'
  926 = 'LIFT ESTOP'
  519 = 'LIFT STATION DETECTION'
  495 = 'LIGHT CURTAIN LEFT'
  39 = 'LIGHT CURTAIN RIGHT'
  413 = 'LOAD'
  897 = 'LOADING SAFETY'
  351 = 'Main'
  386 = 'MCP ESTOP'
  215 = 'mm/s'
  214 = 'mm/s²'
  207 = 'MOVE ABS'
  569 = 'Move relative'
  205 = 'Neg LS'
  677 = 'outbound'
  842 = 'photosensor[0]'
  79 = 'photosensor[1]'
  70 = 'photo_sensor[0]'
  919 = 'photo_sensor[1]'
  800 = 'photo_sensor_mute'
  925 = 'photo_sensor_mute_l'
  891 = 'photo_sensor_start'
  1003 = 'place'
  204 = 'Pos LS'
  844 = 'Power \nOn'
  359 = 'Power On'
  342 = 'ReM'
  1185 = 'ReM3'
  904 = 'ReM4'
  274 = 'ReM5'
  199 = 'Reset'
  10 = 'RESET'
  1651 = 'retract'
  934 = 'retracted'
  71 = 'ROBOT EAS'
  312 = 'ROBOT EES'
  72 = 'roller'
  1437 = 'Roller In'
  189 = 'roller[0]'
  709 = 'roller[1]'
  633 = 'roller[2]'
  687 = 'roller[3]'
  522 = 'roller_x'
  792 = 'roller_y'
  845 = 'RUN'
  634 = 'SAFETY DOOR'
  202 = 'SAFETY INPUT'
  617 = 'SAFETY OUTPUT'
  641 = 'sComponentID'
  438 = 'sComponent_ID'
  358 = 'sComponent_name'
  874 = 'sensor_mute'
  143 = 'sensor_mute_left'
  487 = 'sensor_mute_right'
  622 = 'Set absolute\nencoder as linear'
  454 = 'Set absolute\nencoder as rotation'
  208 = 'Set Point'
  14 = 'Set Pos to 0'
  332 = 'sEventType'
  714 = 'sEvent_MSG'
  245 = 'sID'
  220 = 'sMethod'
  1077 = 'Start'
  22 = 'Starting'
  67 = 'State Model\n%s'
  1356 = 'Station1'
  1785 = 'Station2'
  1034 = 'StepID'
  986 = 'sTime'
  198 = 'Stop'
  996 = 'STOP'
  1671 = 'stop'
  31 = 'Stopped'
  35 = 'Stopping'
  1097 = 'Suspend'
  28 = 'Suspended'
  29 = 'Suspending'
  666 = 'Time'
  2038 = 'time_detection'
  2651 = 'Tote1'
  1283 = 'Tote2'
  784 = 'tote_detection'
  1613 = 'TryRunMode'
  590 = 'TryRunStart'
  118 = 'TryRunStop'
  585 = 'Type'
  13 = 'Unhold'
  24 = 'Unholding'
  20 = 'Unit Mode'
  780 = 'UNLOAD'
  809 = 'Unload'
  2590 = 'Unload To Left'
  297 = 'Unload To Right'
  37 = 'Unsuspend'
  27 = 'Unsuspending'
  15 = 'Unuspend'
  407 = 'UP'
  505 = 'Up'
  848 = 'User'
  8 = 'UserMode 1'
  863 = 'valve_clamp[0]'
  1846 = 'valve_left_door'
  1781 = 'valve_left_door extend'
  2324 = 'valve_left_door valve_left_door.extend'
  676 = 'valve_left_door.extend'
  1741 = 'valve_lif'
  396 = 'valve_lift'
  464 = 'valve_lift[0]'
  247 = 'valve_lift_1'
  1409 = 'valve_lift_2'
  2061 = 'valve_lif_1'
  1819 = 'valve_right_door'
  227 = 'valve_stopper'
  200 = 'Velocity'
  193 = 'WORKING SAFETY'
  246 = 'Working1'
  753 = 'Working1 Load'
  928 = 'Working1 Unload'
  514 = 'Working2'
  2337 = 'Working2 Load'
  86 = 'Working2 Unload'
  1 = 'Yes'
  2 = 'Yes, with Reset'
END_TEXTLIST

// ---- VISUs/Templates/visu_autoStore.TcVIS
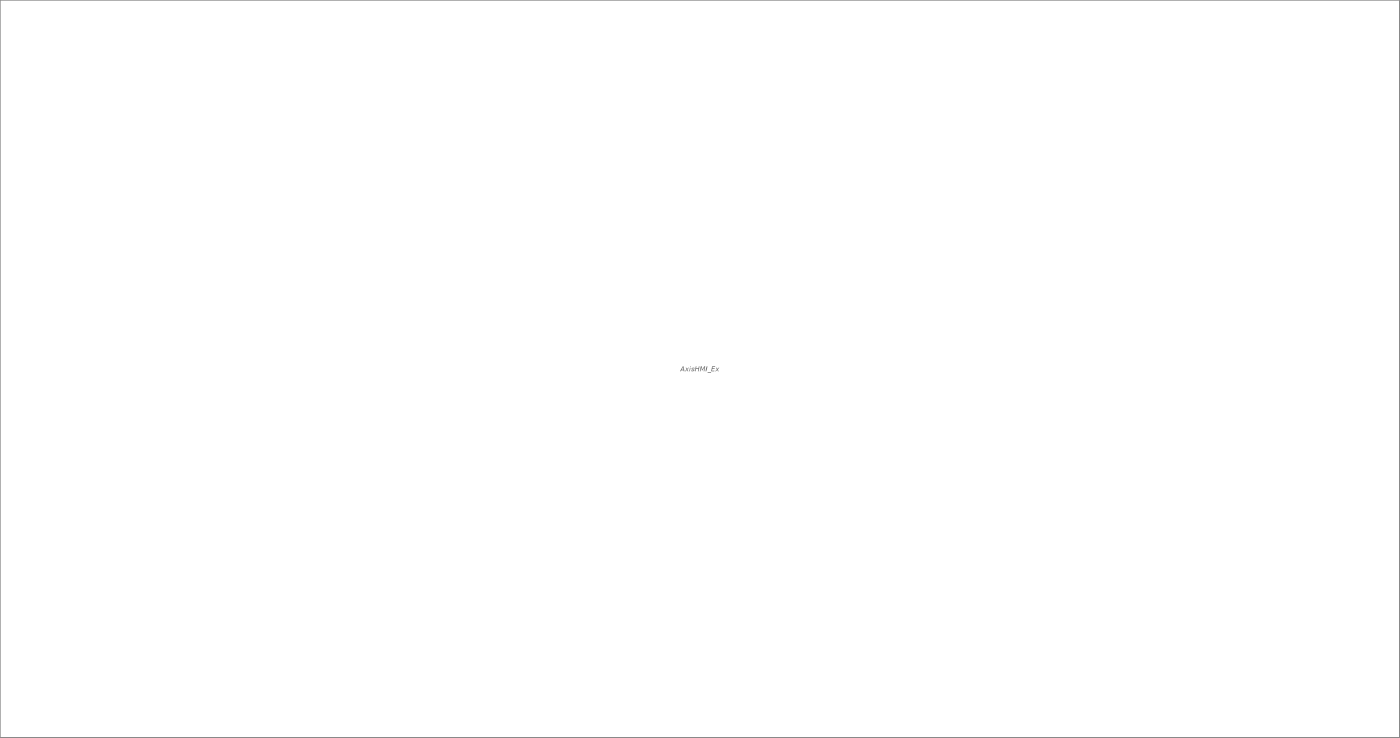
VISUALIZATION visu_autoStore  // 2048x1080
VAR_IN_OUT
	autoStore	: FB_autoStore;
END_VAR
    TabControl (0,0 2048x1080)
        shows AxisHMI_Ex(stAxisHMI := autoStore.st_mcAxis_lift, mcAxis := autoStore.mcAxis_lift, xError := autoStore.mcAxis_lift.xError)
        shows AxisHMI_Ex(stAxisHMI := autoStore.st_mcAxis_transfer, mcAxis := autoStore.mcAxis_transfer, xError := autoStore.mcAxis_transfer.xError)
        shows v_io_autoStore(autoStore := autoStore)
        shows AxisHMI_Ex(stAxisHMI := GVL.fb_working.st_mcAxis_vacuun[0], mcAxis := GVL.fb_working.mcAxis_vacuun[0], xError := GVL.fb_working.mcAxis_vacuun[0].xError)
        shows AxisHMI_Ex(stAxisHMI := GVL.fb_working.st_mcAxis_vacuun[1], mcAxis := GVL.fb_working.mcAxis_vacuun[1], xError := GVL.fb_working.mcAxis_vacuun[1].xError)
        shows AxisHMI_Ex(stAxisHMI := GVL.fb_working.st_mcAxis_bagOpen[0], mcAxis := GVL.fb_working.mcAxis_bagOpen[0], xError := GVL.fb_working.mcAxis_bagOpen[0].xError)
        shows AxisHMI_Ex(stAxisHMI := GVL.fb_working.st_mcAxis_bagOpen[1], mcAxis := GVL.fb_working.mcAxis_bagOpen[1], xError := GVL.fb_working.mcAxis_bagOpen[1].xError)
        shows AxisHMI_Ex(stAxisHMI := GVL.fb_working.st_mcAxis_bagOpen[2], mcAxis := GVL.fb_working.mcAxis_bagOpen[2], xError := GVL.fb_working.mcAxis_bagOpen[2].xError)
        shows AxisHMI_Ex(stAxisHMI := GVL.fb_working.st_mcAxis_bagOpen[3], mcAxis := GVL.fb_working.mcAxis_bagOpen[3], xError := GVL.fb_working.mcAxis_bagOpen[3].xError)
        [0]: TabTitle=Lift
        [1]: TabTitle=BagOpen
        [3]: TabTitle=Axis_vacuun_0
        [4]: TabTitle=Axis_vacuun_1
        [5]: TabTitle=Axis_bagOpen_0
        [6]: TabTitle=Axis_bagOpen_1
        [7]: TabTitle=Axis_bagOpen_2
        [8]: TabTitle=Axis_bagOpen_3
        p2837713833: gantrybase.mcAxis[EN_Axis.Z].sAxisName
END_VISUALIZATION

// ---- VISUs/Templates/VIS_TemplatePMLStateModel.TcVIS
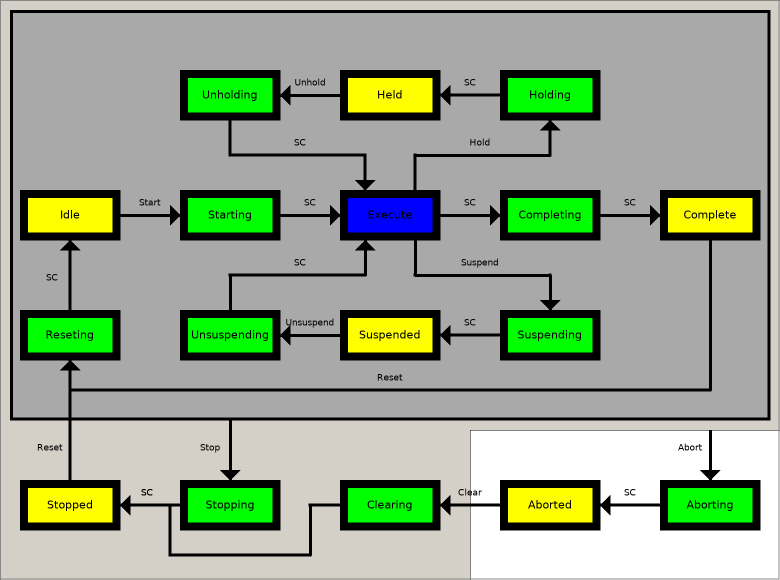
VISUALIZATION VIS_TemplatePMLStateModel  // 780x580
VAR_INPUT
	ePMLUnitMode		: DINT;
	ePMLState			: DINT;
END_VAR
VAR_IN_OUT
	eStateCommand		: DINT;
END_VAR
    Polygon (0,0) (780,0) (780,430) (470,430) (470,580) (0,580)
    Rectangle (10,10 760x410)
    Polyline (415,190) (415,155) (550,155) (550,95) (440,95), invisible if: stPMLUnitModeConfiguration[ePMLUnitMode].aStateDisabled[11]
    Polyline (365,190) (365,155) (230,155) (230,95) (340,95), invisible if: stPMLUnitModeConfiguration[ePMLUnitMode].aStateDisabled[11]
    Polyline (415,240) (415,275) (550,275) (550,335) (440,335), invisible if: stPMLUnitModeConfiguration[ePMLUnitMode].aStateDisabled[5]
    Polyline (365,240) (365,275) (230,275) (230,335) (340,335), invisible if: stPMLUnitModeConfiguration[ePMLUnitMode].aStateDisabled[5]
    Polyline (710,430) (710,505) (310,505) (310,555) (170,555) (170,505) (70,505) (70,215) (340,215)
    RoundedRectangle (20,190 100x50), "Idle", colour toggle: (ePMLState = 4), invisible if: stPMLUnitModeConfiguration[ePMLUnitMode].aStateDisabled[4]
    RoundedRectangle (180,190 100x50), "Starting", colour toggle: (ePMLState = 3), invisible if: stPMLUnitModeConfiguration[ePMLUnitMode].aStateDisabled[3]
    RoundedRectangle (340,190 100x50), "Execute", colour toggle: (ePMLState = 6)
    RoundedRectangle (180,70 100x50), "Unholding", colour toggle: (ePMLState = 12), invisible if: stPMLUnitModeConfiguration[ePMLUnitMode].aStateDisabled[12]
    RoundedRectangle (340,70 100x50), "Held", colour toggle: (ePMLState = 11), invisible if: stPMLUnitModeConfiguration[ePMLUnitMode].aStateDisabled[11]
    RoundedRectangle (500,70 100x50), "Holding", colour toggle: (ePMLState = 10), invisible if: stPMLUnitModeConfiguration[ePMLUnitMode].aStateDisabled[10]
    RoundedRectangle (180,310 100x50), "Unsuspending", colour toggle: (ePMLState = 14), invisible if: stPMLUnitModeConfiguration[ePMLUnitMode].aStateDisabled[14]
    RoundedRectangle (340,310 100x50), "Suspended", colour toggle: (ePMLState = 5), invisible if: stPMLUnitModeConfiguration[ePMLUnitMode].aStateDisabled[5]
    RoundedRectangle (500,310 100x50), "Suspending", colour toggle: (ePMLState = 13), invisible if: stPMLUnitModeConfiguration[ePMLUnitMode].aStateDisabled[13]
    RoundedRectangle (20,310 100x50), "Reseting", colour toggle: (ePMLState = 15), invisible if: stPMLUnitModeConfiguration[ePMLUnitMode].aStateDisabled[15]
    RoundedRectangle (20,480 100x50), "Stopped", colour toggle: (ePMLState = 2)
    RoundedRectangle (340,480 100x50), "Clearing", colour toggle: (ePMLState = 1), invisible if: stPMLUnitModeConfiguration[ePMLUnitMode].aStateDisabled[1]
    RoundedRectangle (500,480 100x50), "Aborted", colour toggle: (ePMLState = 9)
    RoundedRectangle (660,480 100x50), "Aborting", colour toggle: (ePMLState = 8), invisible if: stPMLUnitModeConfiguration[ePMLUnitMode].aStateDisabled[8]
    Polygon (550,120) (540,130) (560,130), invisible if: stPMLUnitModeConfiguration[ePMLUnitMode].aStateDisabled[10]
    Polygon (365,240) (355,250) (375,250), invisible if: stPMLUnitModeConfiguration[ePMLUnitMode].aStateDisabled[5]
    Polygon (70,240) (60,250) (80,250), invisible if: stPMLUnitModeConfiguration[ePMLUnitMode].aStateDisabled[4]
    Polygon (70,360) (60,370) (80,370), invisible if: stPMLUnitModeConfiguration[ePMLUnitMode].aStateDisabled[15]
    Polygon (440,95) (450,105) (450,85), invisible if: stPMLUnitModeConfiguration[ePMLUnitMode].aStateDisabled[11]
    Polygon (280,95) (290,105) (290,85), invisible if: stPMLUnitModeConfiguration[ePMLUnitMode].aStateDisabled[12]
    Polygon (440,335) (450,345) (450,325), invisible if: stPMLUnitModeConfiguration[ePMLUnitMode].aStateDisabled[5]
    Polygon (280,335) (290,345) (290,325), invisible if: stPMLUnitModeConfiguration[ePMLUnitMode].aStateDisabled[14]
    Polygon (600,505) (610,515) (610,495)
    Polygon (440,505) (450,515) (450,495), invisible if: stPMLUnitModeConfiguration[ePMLUnitMode].aStateDisabled[1]
    Polygon (120,505) (130,515) (130,495)
    Polygon (180,215) (170,225) (170,205), invisible if: stPMLUnitModeConfiguration[ePMLUnitMode].aStateDisabled[3]
    Polygon (340,215) (330,225) (330,205)
    Polygon (500,215) (490,225) (490,205), invisible if: stPMLUnitModeConfiguration[ePMLUnitMode].aStateDisabled[16]
    Polygon (660,215) (650,225) (650,205), invisible if: stPMLUnitModeConfiguration[ePMLUnitMode].aStateDisabled[17]
    Polygon (375,180) (365,190) (355,180), invisible if: stPMLUnitModeConfiguration[ePMLUnitMode].aStateDisabled[11]
    Polygon (560,300) (550,310) (540,300), invisible if: stPMLUnitModeConfiguration[ePMLUnitMode].aStateDisabled[13]
    Polygon (720,470) (710,480) (700,470), invisible if: stPMLUnitModeConfiguration[ePMLUnitMode].aStateDisabled[8]
    Polygon (240,470) (230,480) (220,470), invisible if: stPMLUnitModeConfiguration[ePMLUnitMode].aStateDisabled[7]
    Polyline (230,420) (230,505) (150,505)
    RoundedRectangle (180,480 100x50), "Stopping", colour toggle: (ePMLState = 7), invisible if: stPMLUnitModeConfiguration[ePMLUnitMode].aStateDisabled[7]
    Label (440,135 80x15), "Hold", invisible if: stPMLUnitModeConfiguration[ePMLUnitMode].aStateDisabled[11]
    Label (260,135 80x15), "SC", invisible if: stPMLUnitModeConfiguration[ePMLUnitMode].aStateDisabled[12]
    Label (430,75 80x15), "SC", invisible if: stPMLUnitModeConfiguration[ePMLUnitMode].aStateDisabled[10]
    Label (270,75 80x15), "Unhold", invisible if: stPMLUnitModeConfiguration[ePMLUnitMode].aStateDisabled[11]
    Label (270,315 80x15), "Unsuspend", invisible if: stPMLUnitModeConfiguration[ePMLUnitMode].aStateDisabled[5]
    Label (430,315 80x15), "SC", invisible if: stPMLUnitModeConfiguration[ePMLUnitMode].aStateDisabled[13]
    Label (440,255 80x15), "Suspend", invisible if: stPMLUnitModeConfiguration[ePMLUnitMode].aStateDisabled[5]
    Label (260,255 80x15), "SC", invisible if: stPMLUnitModeConfiguration[ePMLUnitMode].aStateDisabled[14]
    Label (270,195 80x15), "SC", invisible if: stPMLUnitModeConfiguration[ePMLUnitMode].aStateDisabled[3]
    Label (590,195 80x15), "SC", invisible if: stPMLUnitModeConfiguration[ePMLUnitMode].aStateDisabled[16]
    Label (430,195 80x15), "SC", invisible if: stPMLUnitModeConfiguration[ePMLUnitMode].aStateDisabled[17]
    Label (430,485 80x15), "Clear"
    Label (590,485 80x15), "SC", invisible if: stPMLUnitModeConfiguration[ePMLUnitMode].aStateDisabled[8]
    Label (107,485 80x15), "SC", invisible if: stPMLUnitModeConfiguration[ePMLUnitMode].aStateDisabled[1]
    Label (350,370 80x15), "Reset", invisible if: stPMLUnitModeConfiguration[ePMLUnitMode].aStateDisabled[17]
    Label (10,440 80x15), "Reset", invisible if: stPMLUnitModeConfiguration[ePMLUnitMode].aStateDisabled[4]
    Label (170,440 80x15), "Stop"
    Label (650,440 80x15), "Abort"
    Label (12,270 80x15), "SC", invisible if: stPMLUnitModeConfiguration[ePMLUnitMode].aStateDisabled[15]
    Label (110,195 80x15), "Start"
    Label (107,485 80x15), "SC", invisible if: stPMLUnitModeConfiguration[ePMLUnitMode].aStateDisabled[7]
    Polyline (440,215) (710,215) (710,390) (70,390), invisible if: stPMLUnitModeConfiguration[ePMLUnitMode].aStateDisabled[17]
    RoundedRectangle (660,190 100x50), "Complete", colour toggle: (ePMLState = 17), invisible if: stPMLUnitModeConfiguration[ePMLUnitMode].aStateDisabled[17]
    RoundedRectangle (500,190 100x50), "Completing", colour toggle: (ePMLState = 16), invisible if: stPMLUnitModeConfiguration[ePMLUnitMode].aStateDisabled[16]
END_VISUALIZATION

// ---- VISUs/Templates/v_io_autoStore.TcVIS
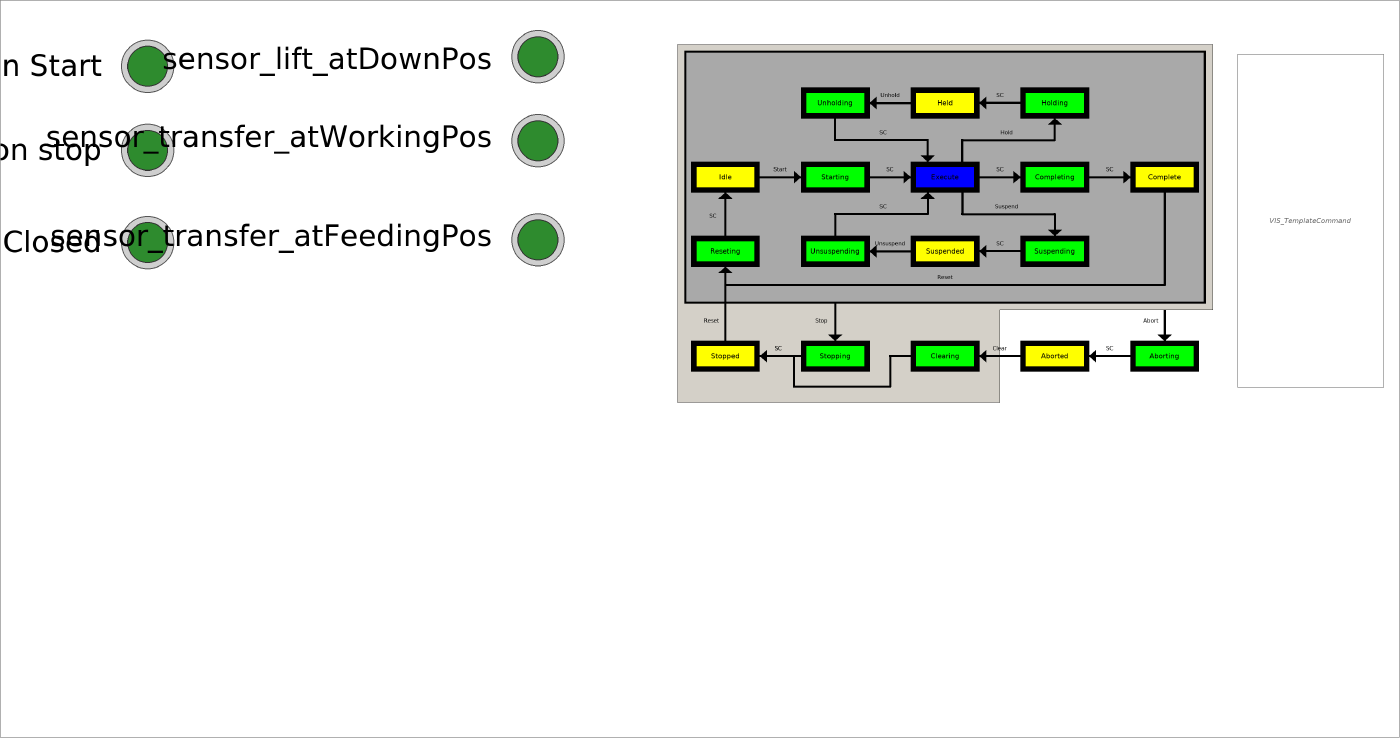
VISUALIZATION v_io_autoStore  // 2048x1080
VAR_IN_OUT
	autoStore	: FB_autoStore;
END_VAR
    Lamp1 (171,52 90x90), variable: autoStore.button_start, style: Lamp-Lamp1-Green
    Label (32,51 120x90), "Btton Start"
    Lamp1 (171,175 90x90), variable: autoStore.button_stop, style: Lamp-Lamp1-Green
    Label (32,174 120x90), "Button stop"
    Lamp1 (171,310 90x90), variable: autoStore.door_closed, style: Lamp-Lamp1-Green
    Label (32,309 120x90), "Door Closed"
    Lamp1 (742,38 90x90), variable: autoStore.sensor_lift_atDownPos, style: Lamp-Lamp1-Green
    Label (409,52 314x68), "sensor_lift_atDownPos"
    Lamp1 (742,161 90x90), variable: autoStore.sensor_transfer_atWorkingPos, style: Lamp-Lamp1-Green
    Label (339,170 384x60), "sensor_transfer_atWorkingPos"
    Lamp1 (742,306 90x90), variable: autoStore.sensor_transfer_atFeedingPos, style: Lamp-Lamp1-Green
    Label (339,315 384x60), "sensor_transfer_atFeedingPos"
    Frame (991,65 783x524)
        shows VIS_TemplatePMLStateModel(ePMLUnitMode := MAIN.fbVisu.eModeVisu, ePMLState := GVL.fb_autoStore1.eState, eStateCommand := MAIN.fbVisu.eUnitCommand)
        shows VIS_TemplatePMLStateModel()
    Frame (1810,79 214x488)
        shows VIS_TemplateCommand(eModeCommand := GVL.PackTags.Command.UnitMode, eStateCommand := GVL.PackTags1.Command.CntrlCmd, eModeStatus := GVL.PackTags.Status.UnitModeCurrent, eStateStatus := GVL.PackTags1.Status.StateCurrent, bModeChangeReq := GVL.PackTags.Command.UnitModeChangeRequest)
END_VISUALIZATION

// ---- VISUs/VISUs/visu_2sys.TcVIS
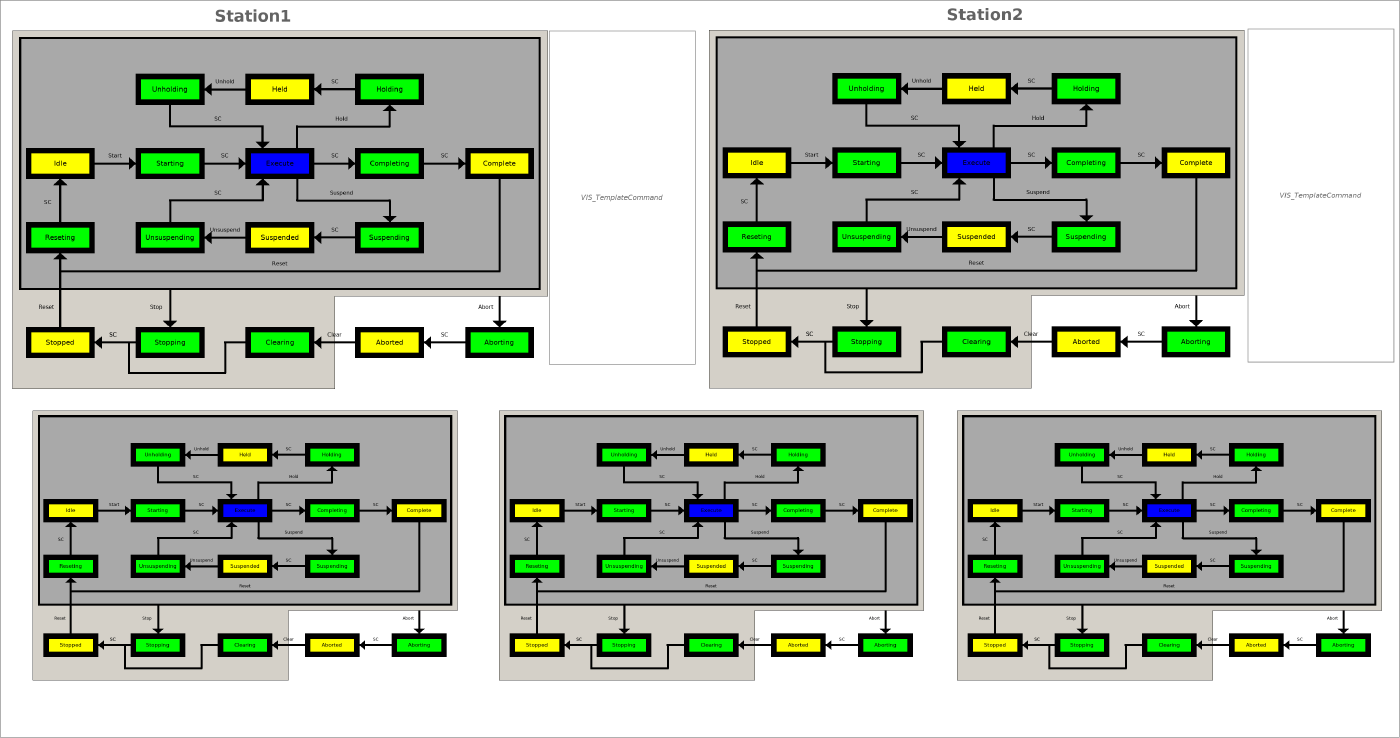
VISUALIZATION visu_2sys  // 2048x1080
    Frame (803,45 214x488)
        shows VIS_TemplateCommand(eModeCommand := GVL.PackTags.Command.UnitMode, eStateCommand := GVL.PackTags1.Command.CntrlCmd, eModeStatus := GVL.PackTags.Status.UnitModeCurrent, eStateStatus := GVL.PackTags1.Status.StateCurrent, bModeChangeReq := GVL.PackTags.Command.UnitModeChangeRequest)
    Frame (1825,42 214x488)
        shows VIS_TemplateCommand(eModeCommand := GVL.PackTags.Command.UnitMode, eStateCommand := GVL.PackTags2.Command.CntrlCmd, eModeStatus := GVL.PackTags.Status.UnitModeCurrent, eStateStatus := GVL.PackTags2.Status.StateCurrent, bModeChangeReq := GVL.PackTags.Command.UnitModeChangeRequest)
    Frame (18,45 783x524)
        shows VIS_TemplatePMLStateModel(ePMLUnitMode := MAIN.fbVisu.eModeVisu, ePMLState := MAIN.fbMachine1.eState, eStateCommand := MAIN.fbVisu.eUnitCommand)
        shows VIS_TemplatePMLStateModel()
    Frame (1037,44 783x524)
        shows VIS_TemplatePMLStateModel(ePMLUnitMode := MAIN.fbVisu.eModeVisu, ePMLState := MAIN.fbMachine2.eState, eStateCommand := MAIN.fbVisu.eUnitCommand)
        shows VIS_TemplatePMLStateModel()
    Frame (48,601 621x394)
        shows VIS_TemplatePMLStateModel(ePMLUnitMode := MAIN.fbVisu.eModeVisu, ePMLState := GVL.fb_working1.eState, eStateCommand := MAIN.fbVisu.eUnitCommand)
        shows VIS_TemplatePMLStateModel()
    Frame (730,601 621x394)
        shows VIS_TemplatePMLStateModel(ePMLUnitMode := MAIN.fbVisu.eModeVisu, ePMLState := GVL.fb_loading.eState, eStateCommand := MAIN.fbVisu.eUnitCommand)
        shows VIS_TemplatePMLStateModel()
    Frame (1400,601 621x394)
        shows VIS_TemplatePMLStateModel(ePMLUnitMode := MAIN.fbVisu.eModeVisu, ePMLState := GVL.fb_working2.eState, eStateCommand := MAIN.fbVisu.eUnitCommand)
        shows VIS_TemplatePMLStateModel()
    Label (295,1 150x45), "Station1"
    Label (1366,-1 150x45), "Station2"
END_VISUALIZATION

// ---- VISUs/VISUs/visu_operation.TcVIS
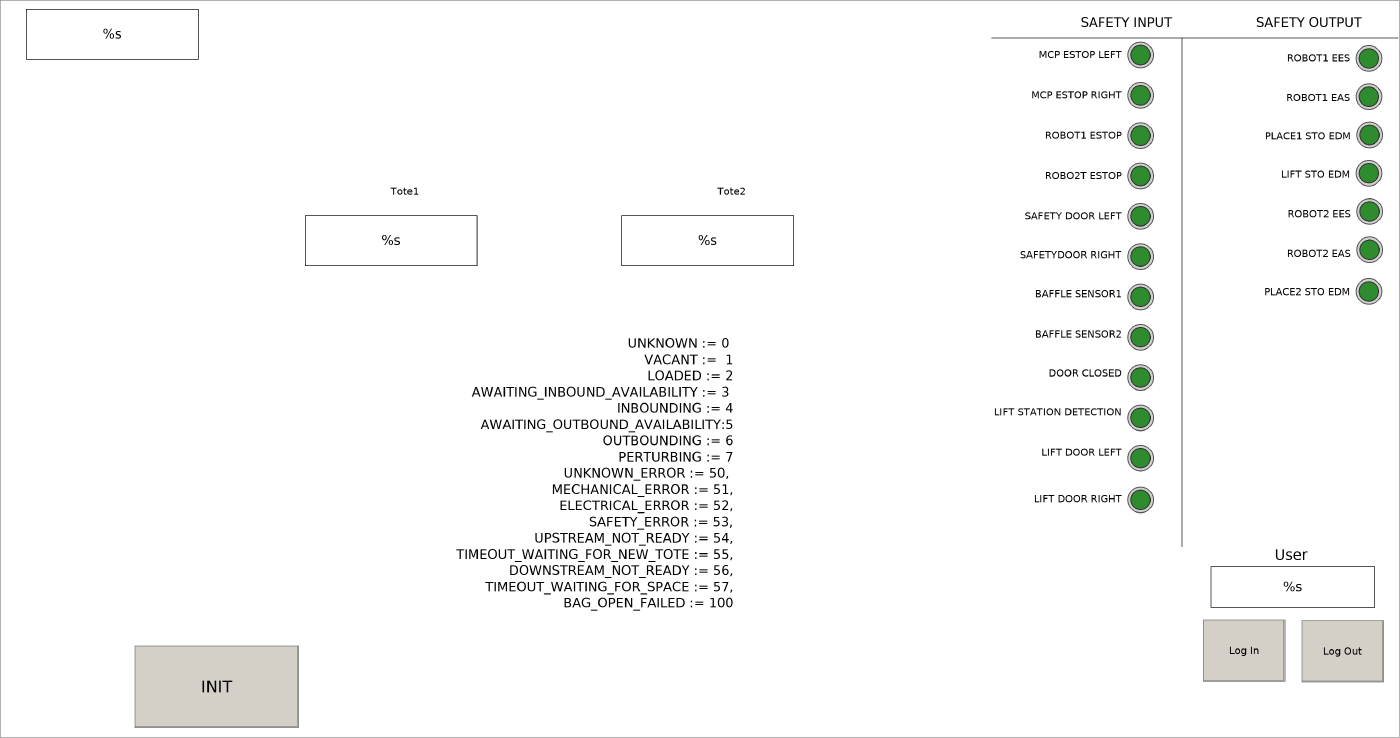
VISUALIZATION visu_operation  // 2048x1080
    Button (197,945 240x120), "INIT", colour toggle: G_HMI.bInit
        OnMouseDown: execute { G_HMI.bInit	:= TRUE; }
        OnMouseUp: execute { G_HMI.bInit	:= FALSE; }
    Lamp1 (1646,58 45x45), variable: MAIN.safety_1.mcp_estop_left.Q, style: Lamp-Lamp1-Green
    Label (1344,65 300x30), "MCP ESTOP LEFT"
    Lamp1 (1646,117 45x45), variable: MAIN.safety_1.mcp_estop_right.Q, style: Lamp-Lamp1-Green
    Label (1344,124 300x30), "MCP ESTOP RIGHT"
    Lamp1 (1646,353 45x45), variable: MAIN.safety_1.safetyDoor_right, style: Lamp-Lamp1-Green
    Label (1344,360 300x26), "SAFETYDOOR RIGHT"
    Lamp1 (1646,530 45x45), variable: MAIN.safety_1.door_closed, style: Lamp-Lamp1-Green
    Label (1344,533 300x26), "DOOR CLOSED"
    Lamp1 (1646,589 45x45), variable: MAIN.safety_1.lift_station_detection, style: Lamp-Lamp1-Green
    Label (1344,588 300x30), "LIFT STATION DETECTION"
    Lamp1 (1980,63 45x45), variable: GVL_SAFETY.robot1_STO_EES, style: Lamp-Lamp1-Green
    Label (1728,70 250x30), "ROBOT1 EES"
    Lamp1 (1980,231 45x45), variable: GVL_SAFETY.Lift_STO, style: Lamp-Lamp1-Green
    Label (1728,240 250x30), "LIFT STO EDM"
    Lamp1 (1981,175 45x45), variable: GVL_SAFETY.Place1_STO, style: Lamp-Lamp1-Green
    Label (1729,186 250x26), "PLACE1 STO EDM"
    Lamp1 (1980,404 45x45), variable: GVL_SAFETY.Place2_STO, style: Lamp-Lamp1-Green
    Label (1728,414 250x26), "PLACE2 STO EDM"
    Lamp1 (1980,119 45x45), variable: GVL_SAFETY.robot1_STO_EAS, style: Lamp-Lamp1-Green
    Label (1728,128 250x30), "ROBOT1 EAS"
    Line (1729,800) (1729,55)
    Label (1523,18 250x30), "SAFETY INPUT"
    Label (1790,18 250x30), "SAFETY OUTPUT"
    Line (1450,55) (2045,55)
    Rectangle (38,13 252x74), "%s"
    Rectangle (1771,829 240x60), "%s", text variable: G_HMI.sLoginnedUser
    Button (1904,908 120x90), "Log Out"
        OnMouseDown: VisuUserMgmt Type=Logout
    Button (1760,907 120x90), "Log In"
        OnMouseDown: VisuUserMgmt Type=Login
    Label (1814,797 150x30), "User"
    Label (1344,647 300x30), "LIFT DOOR LEFT"
    Lamp1 (1646,648 45x45), variable: MAIN.safety_1.lift_door_left.Q, style: Lamp-Lamp1-Green
    Label (1344,715 300x30), "LIFT DOOR RIGHT"
    Lamp1 (1646,709 45x45), variable: MAIN.safety_1.lift_door_right.Q, style: Lamp-Lamp1-Green
    Label (1344,301 300x30), "SAFETY DOOR LEFT"
    Lamp1 (1646,294 45x45), variable: MAIN.safety_1.safetyDoor_left, style: Lamp-Lamp1-Green
    Label (1344,415 300x30), "BAFFLE SENSOR1"
    Lamp1 (1646,412 45x45), variable: MAIN.safety_1.baffle_sensor_1, style: Lamp-Lamp1-Green
    Label (1344,474 300x30), "BAFFLE SENSOR2"
    Lamp1 (1646,471 45x45), variable: MAIN.safety_1.baffle_sensor_2, style: Lamp-Lamp1-Green
    Lamp1 (1981,287 45x45), variable: GVL_SAFETY.robot2_STO_EES, style: Lamp-Lamp1-Green
    Label (1729,298 250x30), "ROBOT2 EES"
    Lamp1 (1981,343 45x45), variable: GVL_SAFETY.robot2_STO_EAS, style: Lamp-Lamp1-Green
    Label (1729,356 250x30), "ROBOT2 EAS"
    Lamp1 (1646,176 45x45), variable: MAIN.safety_1.bRobot1_eStop, style: Lamp-Lamp1-Green
    Label (1344,183 300x30), "ROBOT1 ESTOP"
    Lamp1 (1646,235 45x45), variable: MAIN.safety_1.bRobot2_eStop, style: Lamp-Lamp1-Green
    Label (1344,242 300x30), "ROBO2T ESTOP"
    Label (316,265 300x30), "Tote1"
    Rectangle (446,315 252x74), "%s", text variable: GVL.fb_working1.tote_status
    Label (314,457 762x471), "UNKNOWN := 0 VACANT := 1 LOADED := 2 AWAITING_INBOUND_AVAILABILITY := 3 INBOUNDING := 4 AWAITING_OUTBOUND_AVAILABILITY:5 OUTBOUNDING := 6 PERTURBING := 7 UNKNOWN_ERROR := 50, MECHANICAL_ERROR := 51, ELECTRICAL_ERROR := 52, SAFETY_ERROR := 53, UPSTREAM_NOT_READY := 54, TIMEOUT_WAITING_FOR_NEW_TOTE := 55, DOWNSTREAM_NOT_READY := 56, TIMEOUT_WAITING_FOR_SPACE := 57, BAG_OPEN_FAILED := 100"
    Rectangle (909,315 252x74), "%s", text variable: GVL.fb_working2.tote_status
    Label (794,265 300x30), "Tote2"
END_VISUALIZATION

// ---- VISUs/VISUs/visu_manual.TcVIS
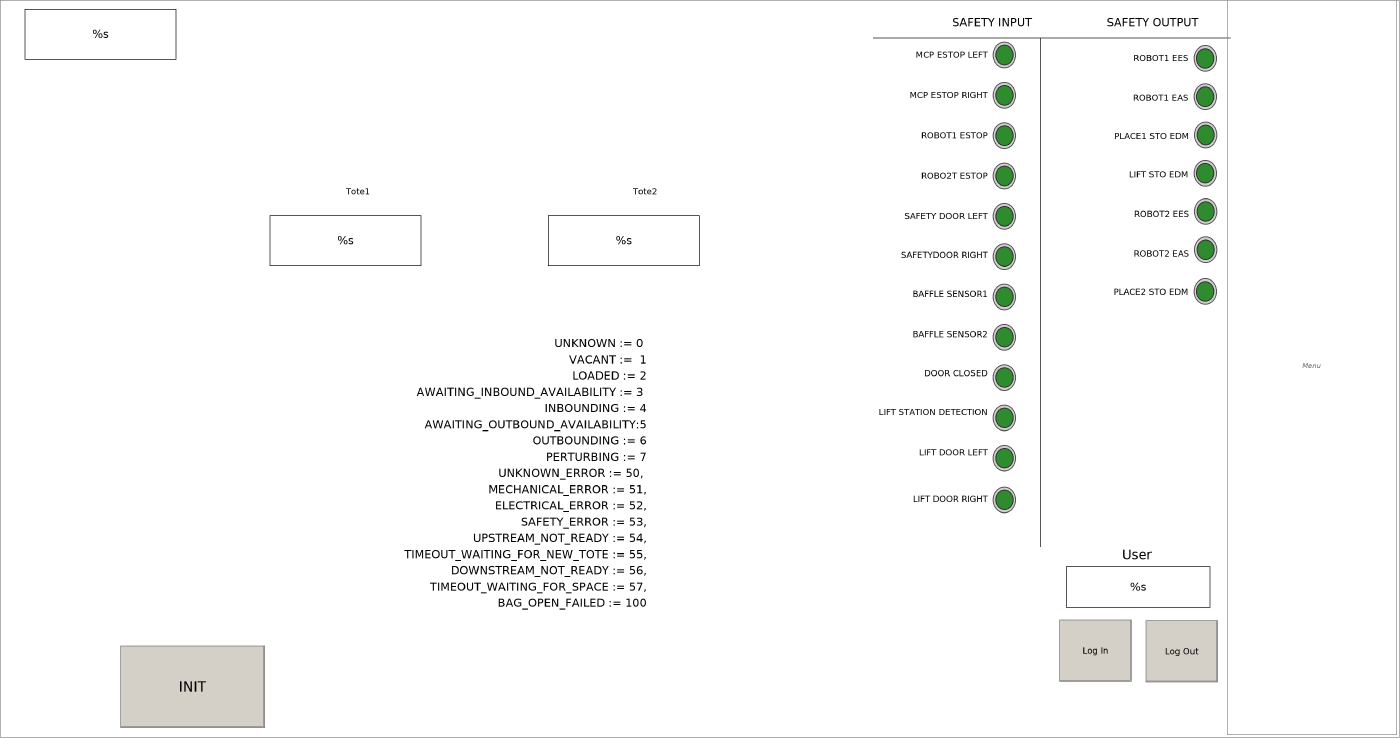
VISUALIZATION visu_manual  // 2048x1080
    Frame (3,0 1800x1080), frame switch variable: G_HMI.iMainFrame
        shows visu_operation()
        shows v_alarm()
        shows visu_loading()
        shows visu_working1()
        shows visu_working2()
        shows visu_2sys()
    Frame (1795,-5 248x1080), frame switch variable: G_HMI.iMainFrame
        shows Menu()
        shows visu_working()
        shows v_IO_fixtureClamp()
        shows visu_buffer()
        shows visu_loading()
        shows v_alarm()
END_VISUALIZATION

// ---- VISUs/VISUs/visu_working1.TcVIS
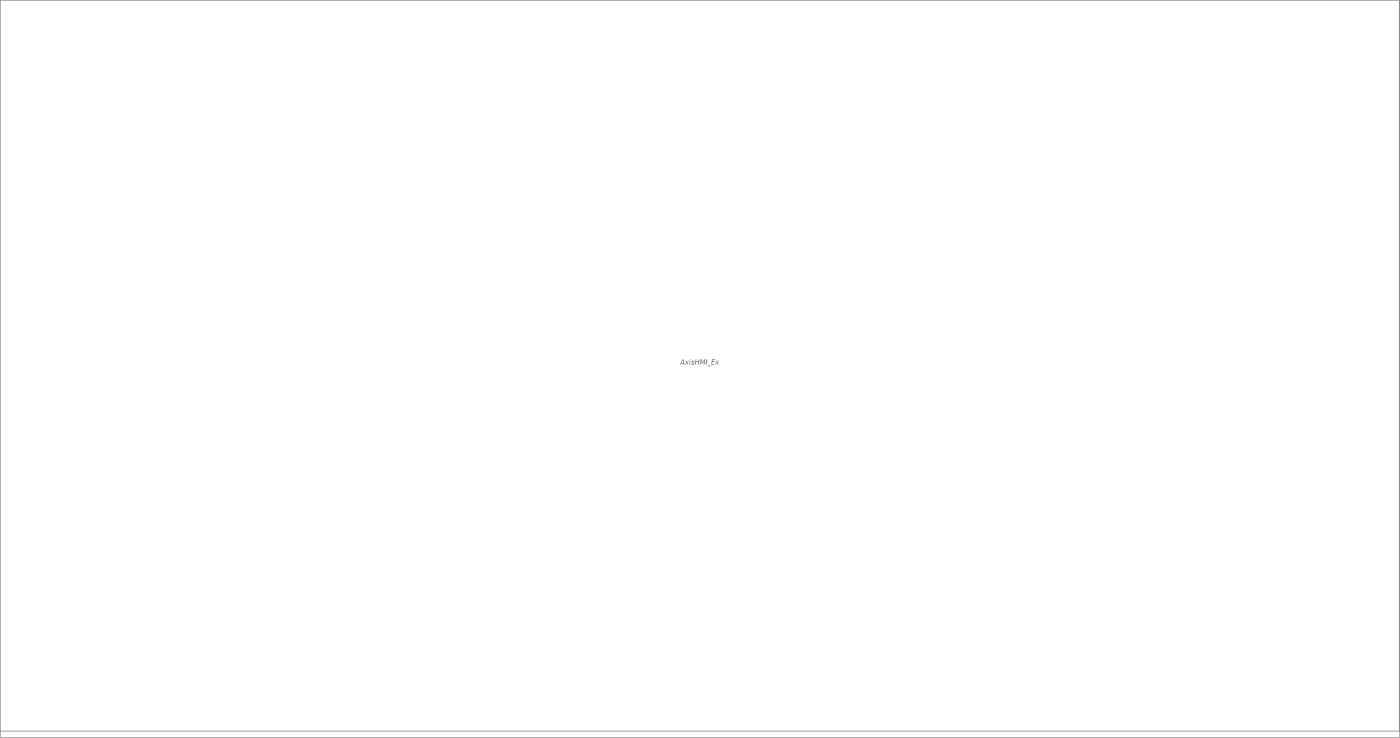
VISUALIZATION visu_working1  // 2048x1080
    TabControl (0,-10 2048x1080)
        shows AxisHMI_Ex(stAxisHMI := GVL.fb_working1.st_mcAxis_lift, mcAxis := GVL.fb_working1.mcAxis_lift, xError := GVL.fb_working1.mcAxis_lift.xError)
        shows AxisHMI_Ex(stAxisHMI := GVL.fb_working1.st_mcAxis_bag, mcAxis := GVL.fb_working1.mcAxis_bag, xError := GVL.fb_working1.mcAxis_bag.xError)
        shows v_io_working1()
        shows AxisHMI_Ex(stAxisHMI := GVL.fb_working.st_mcAxis_vacuun[0], mcAxis := GVL.fb_working.mcAxis_vacuun[0], xError := GVL.fb_working.mcAxis_vacuun[0].xError)
        shows AxisHMI_Ex(stAxisHMI := GVL.fb_working.st_mcAxis_vacuun[1], mcAxis := GVL.fb_working.mcAxis_vacuun[1], xError := GVL.fb_working.mcAxis_vacuun[1].xError)
        shows AxisHMI_Ex(stAxisHMI := GVL.fb_working.st_mcAxis_bagOpen[0], mcAxis := GVL.fb_working.mcAxis_bagOpen[0], xError := GVL.fb_working.mcAxis_bagOpen[0].xError)
        shows AxisHMI_Ex(stAxisHMI := GVL.fb_working.st_mcAxis_bagOpen[1], mcAxis := GVL.fb_working.mcAxis_bagOpen[1], xError := GVL.fb_working.mcAxis_bagOpen[1].xError)
        shows AxisHMI_Ex(stAxisHMI := GVL.fb_working.st_mcAxis_bagOpen[2], mcAxis := GVL.fb_working.mcAxis_bagOpen[2], xError := GVL.fb_working.mcAxis_bagOpen[2].xError)
        shows AxisHMI_Ex(stAxisHMI := GVL.fb_working.st_mcAxis_bagOpen[3], mcAxis := GVL.fb_working.mcAxis_bagOpen[3], xError := GVL.fb_working.mcAxis_bagOpen[3].xError)
        [0]: TabTitle=Lift
        [1]: TabTitle=BagOpen
        [3]: TabTitle=Axis_vacuun_0
        [4]: TabTitle=Axis_vacuun_1
        [5]: TabTitle=Axis_bagOpen_0
        [6]: TabTitle=Axis_bagOpen_1
        [7]: TabTitle=Axis_bagOpen_2
        [8]: TabTitle=Axis_bagOpen_3
        p2837713833: gantrybase.mcAxis[EN_Axis.Z].sAxisName
END_VISUALIZATION

// ---- VISUs/VISUs/visu_autoStore1.TcVIS
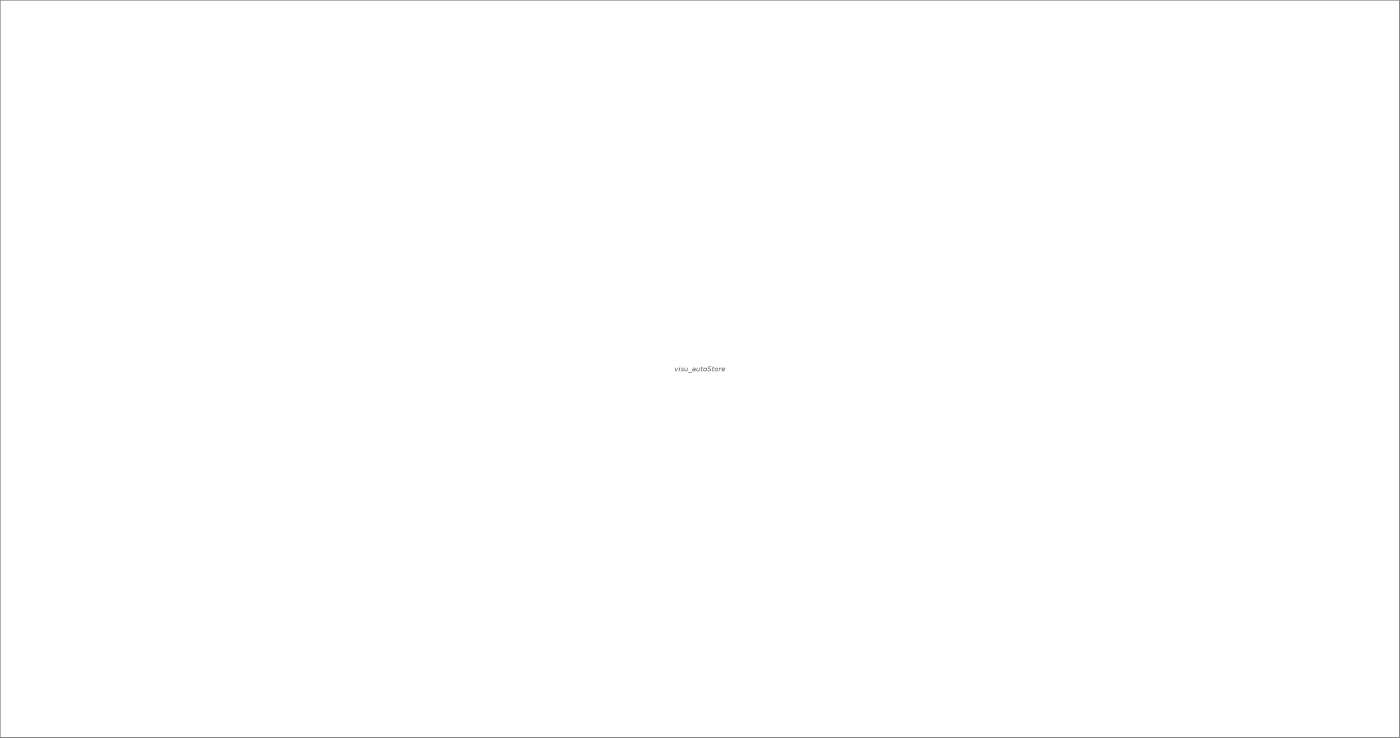
VISUALIZATION visu_autoStore1  // 2048x1080
    TabControl (0,0 2048x1080)
        shows visu_autoStore(autoStore := GVL.fb_autoStore1)
        shows AxisHMI_Ex(stAxisHMI := GVL.fb_working.st_mcAxis_vacuun[0], mcAxis := GVL.fb_working.mcAxis_vacuun[0], xError := GVL.fb_working.mcAxis_vacuun[0].xError)
        shows AxisHMI_Ex(stAxisHMI := GVL.fb_working.st_mcAxis_vacuun[1], mcAxis := GVL.fb_working.mcAxis_vacuun[1], xError := GVL.fb_working.mcAxis_vacuun[1].xError)
        shows AxisHMI_Ex(stAxisHMI := GVL.fb_working.st_mcAxis_bagOpen[0], mcAxis := GVL.fb_working.mcAxis_bagOpen[0], xError := GVL.fb_working.mcAxis_bagOpen[0].xError)
        shows AxisHMI_Ex(stAxisHMI := GVL.fb_working.st_mcAxis_bagOpen[1], mcAxis := GVL.fb_working.mcAxis_bagOpen[1], xError := GVL.fb_working.mcAxis_bagOpen[1].xError)
        shows AxisHMI_Ex(stAxisHMI := GVL.fb_working.st_mcAxis_bagOpen[2], mcAxis := GVL.fb_working.mcAxis_bagOpen[2], xError := GVL.fb_working.mcAxis_bagOpen[2].xError)
        shows AxisHMI_Ex(stAxisHMI := GVL.fb_working.st_mcAxis_bagOpen[3], mcAxis := GVL.fb_working.mcAxis_bagOpen[3], xError := GVL.fb_working.mcAxis_bagOpen[3].xError)
        shows AxisHMI_Ex(stAxisHMI := GVL.fb_working1.st_mcAxis_bag, mcAxis := GVL.fb_working1.mcAxis_bag, xError := GVL.fb_working1.mcAxis_bag.xError)
        shows v_io_working1()
        [3]: TabTitle=Axis_vacuun_0
        [4]: TabTitle=Axis_vacuun_1
        [5]: TabTitle=Axis_bagOpen_0
        [6]: TabTitle=Axis_bagOpen_1
        [7]: TabTitle=Axis_bagOpen_2
        [8]: TabTitle=Axis_bagOpen_3
        [1]: TabTitle=BagOpen
        p2837713833: gantrybase.mcAxis[EN_Axis.Z].sAxisName
END_VISUALIZATION

// ---- VISUs/VISUs/visu_working2.TcVIS
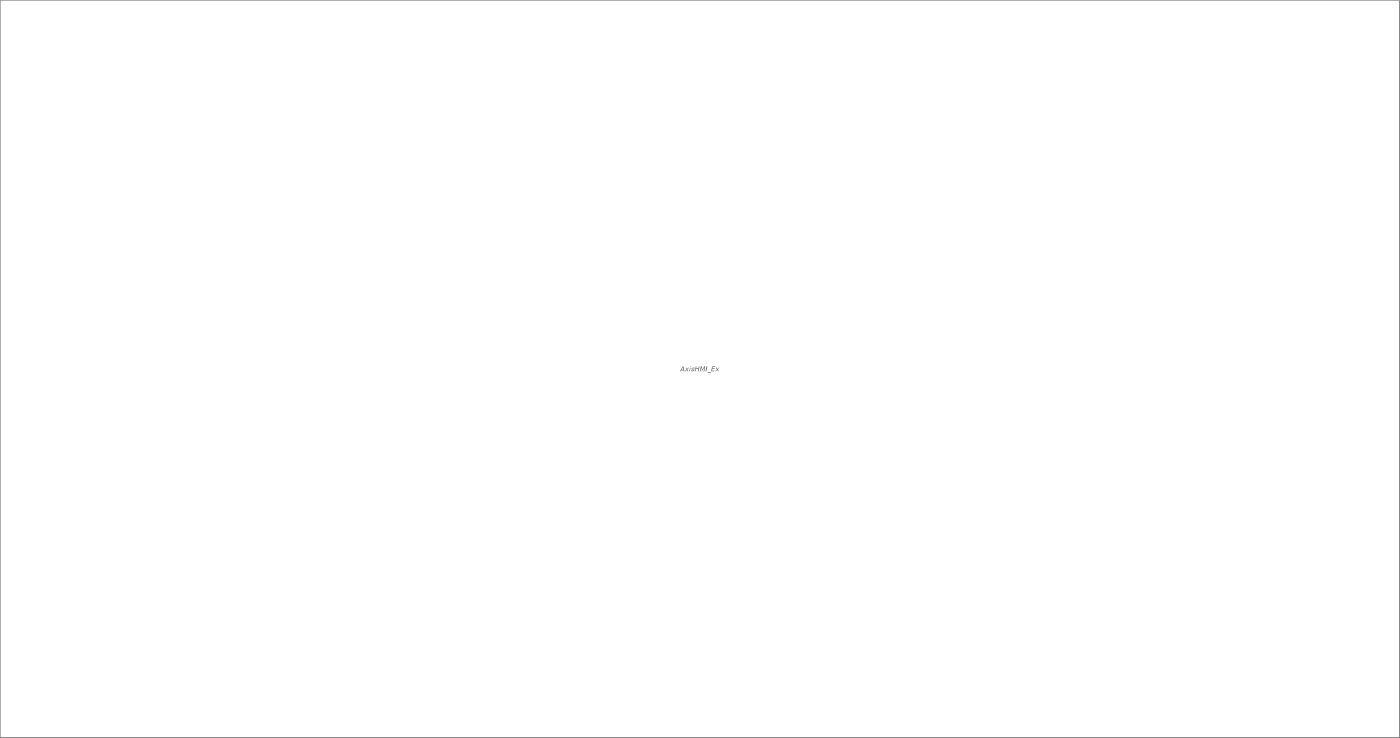
VISUALIZATION visu_working2  // 2048x1080
    TabControl (0,0 2048x1080)
        shows AxisHMI_Ex(stAxisHMI := GVL.fb_working2.st_mcAxis_lift, mcAxis := GVL.fb_working2.mcAxis_lift, xError := GVL.fb_working2.mcAxis_lift.xError)
        shows AxisHMI_Ex(stAxisHMI := GVL.fb_working2.st_mcAxis_bag, mcAxis := GVL.fb_working2.mcAxis_bag, xError := GVL.fb_working2.mcAxis_bag.xError)
        shows v_io_working2()
        shows AxisHMI_Ex(stAxisHMI := GVL.fb_working.st_mcAxis_vacuun[0], mcAxis := GVL.fb_working.mcAxis_vacuun[0], xError := GVL.fb_working.mcAxis_vacuun[0].xError)
        shows AxisHMI_Ex(stAxisHMI := GVL.fb_working.st_mcAxis_vacuun[1], mcAxis := GVL.fb_working.mcAxis_vacuun[1], xError := GVL.fb_working.mcAxis_vacuun[1].xError)
        shows AxisHMI_Ex(stAxisHMI := GVL.fb_working.st_mcAxis_bagOpen[0], mcAxis := GVL.fb_working.mcAxis_bagOpen[0], xError := GVL.fb_working.mcAxis_bagOpen[0].xError)
        shows AxisHMI_Ex(stAxisHMI := GVL.fb_working.st_mcAxis_bagOpen[1], mcAxis := GVL.fb_working.mcAxis_bagOpen[1], xError := GVL.fb_working.mcAxis_bagOpen[1].xError)
        shows AxisHMI_Ex(stAxisHMI := GVL.fb_working.st_mcAxis_bagOpen[2], mcAxis := GVL.fb_working.mcAxis_bagOpen[2], xError := GVL.fb_working.mcAxis_bagOpen[2].xError)
        shows AxisHMI_Ex(stAxisHMI := GVL.fb_working.st_mcAxis_bagOpen[3], mcAxis := GVL.fb_working.mcAxis_bagOpen[3], xError := GVL.fb_working.mcAxis_bagOpen[3].xError)
        [0]: TabTitle=Lift
        [1]: TabTitle=BagOpen
        [3]: TabTitle=Axis_vacuun_0
        [4]: TabTitle=Axis_vacuun_1
        [5]: TabTitle=Axis_bagOpen_0
        [6]: TabTitle=Axis_bagOpen_1
        [7]: TabTitle=Axis_bagOpen_2
        [8]: TabTitle=Axis_bagOpen_3
        p2837713833: gantrybase.mcAxis[EN_Axis.Z].sAxisName
END_VISUALIZATION

// ---- VISUs/VISUs/v_alarm.TcVIS
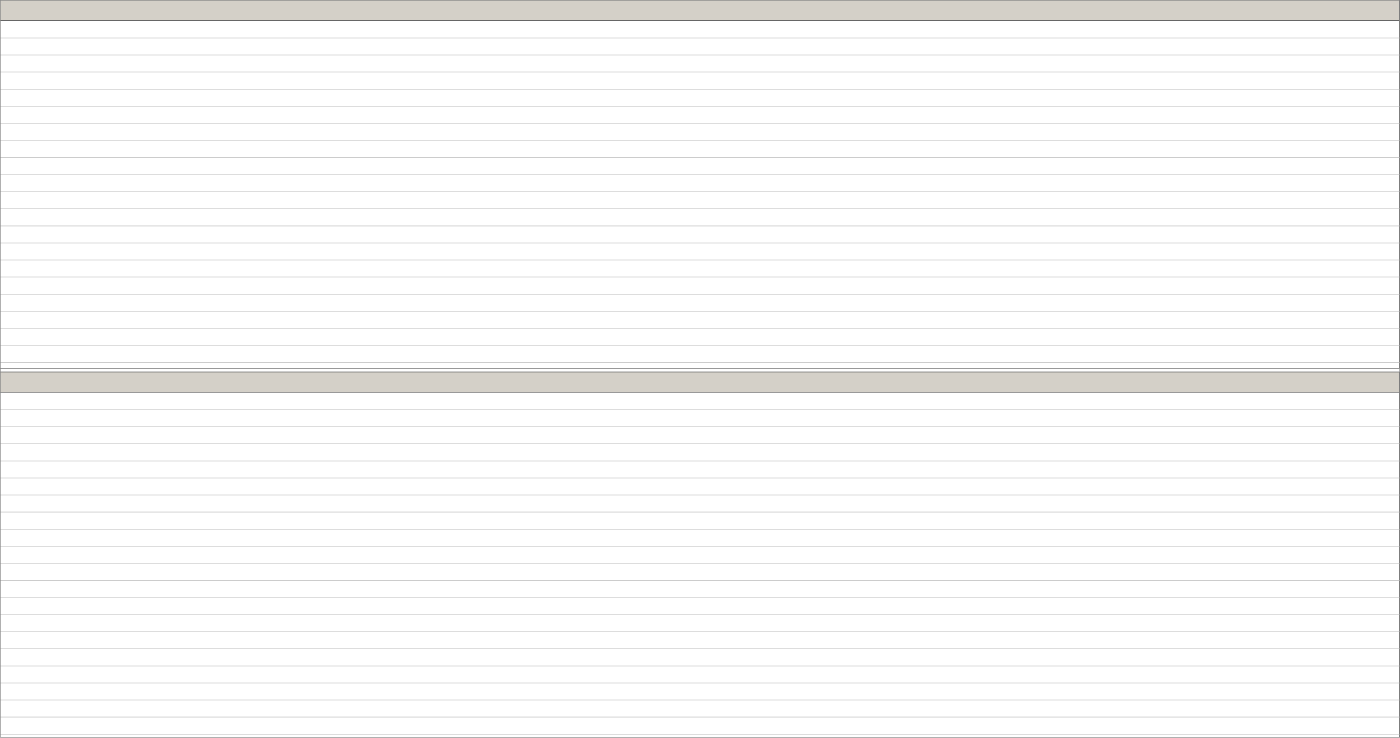
VISUALIZATION v_alarm  // 2048x1080
    Table (0,0 2048x539), data array: GVL.alarms1_hmi
        p3104783080: GVL.fb_buffer.fb_rollers[INDEX].AxisRef
        p2501879983: GVL.fb_buffer.fb_rollers[INDEX].current_tote_status
        p7306298: GVL.fb_buffer.fb_rollers[INDEX].ton_timeout
        p1933151965: GVL.fb_buffer.fb_rollers[INDEX].eStates
        p3863566920: GVL.fb_buffer.fb_rollers[INDEX].iStateTemp
        p2192122294: GVL.fb_buffer.fb_rollers[INDEX].errorMessage
        p400160035: GVL.fb_buffer.fb_rollers[INDEX].xError
        p1265227338: GVL.fb_buffer.fb_rollers[INDEX].rPos_up
        p3726181087: GVL.fb_buffer.fb_rollers[INDEX].rPos_down
        p3854506369: GVL.alarms1_hmi[INDEX].msg
        p1892666644: GVL.alarms1_hmi[INDEX].str_DT
        p338671338: GVL.PackTags.Admin.Alarm[INDEX].Value
        p2170511999: GVL.PackTags.Admin.Alarm[INDEX].Message
        p3723444502: GVL.PackTags.Admin.Alarm[INDEX].Category
        p1218418051: GVL.PackTags.Admin.Alarm[INDEX].DateTime
        p746581629: GVL.PackTags.Admin.Alarm[INDEX].AckDateTime
        p511219082: Datetime
    Table (0,544 2048x535), data array: GVL.alarms2_hmi
        p3104783080: GVL.fb_buffer.fb_rollers[INDEX].AxisRef
        p2501879983: GVL.fb_buffer.fb_rollers[INDEX].current_tote_status
        p7306298: GVL.fb_buffer.fb_rollers[INDEX].ton_timeout
        p1933151965: GVL.fb_buffer.fb_rollers[INDEX].eStates
        p3863566920: GVL.fb_buffer.fb_rollers[INDEX].iStateTemp
        p2192122294: GVL.fb_buffer.fb_rollers[INDEX].errorMessage
        p400160035: GVL.fb_buffer.fb_rollers[INDEX].xError
        p1265227338: GVL.fb_buffer.fb_rollers[INDEX].rPos_up
        p3726181087: GVL.fb_buffer.fb_rollers[INDEX].rPos_down
        p3854506369: GVL.alarms2_hmi[INDEX].msg
        p1892666644: GVL.alarms2_hmi[INDEX].str_DT
        p338671338: GVL.PackTags.Admin.Alarm[INDEX].Value
        p2170511999: GVL.PackTags.Admin.Alarm[INDEX].Message
        p3723444502: GVL.PackTags.Admin.Alarm[INDEX].Category
        p1218418051: GVL.PackTags.Admin.Alarm[INDEX].DateTime
        p746581629: GVL.PackTags.Admin.Alarm[INDEX].AckDateTime
        p511219082: Datetime
END_VISUALIZATION

// ---- VISUs/VISUs/v_io_working1.TcVIS
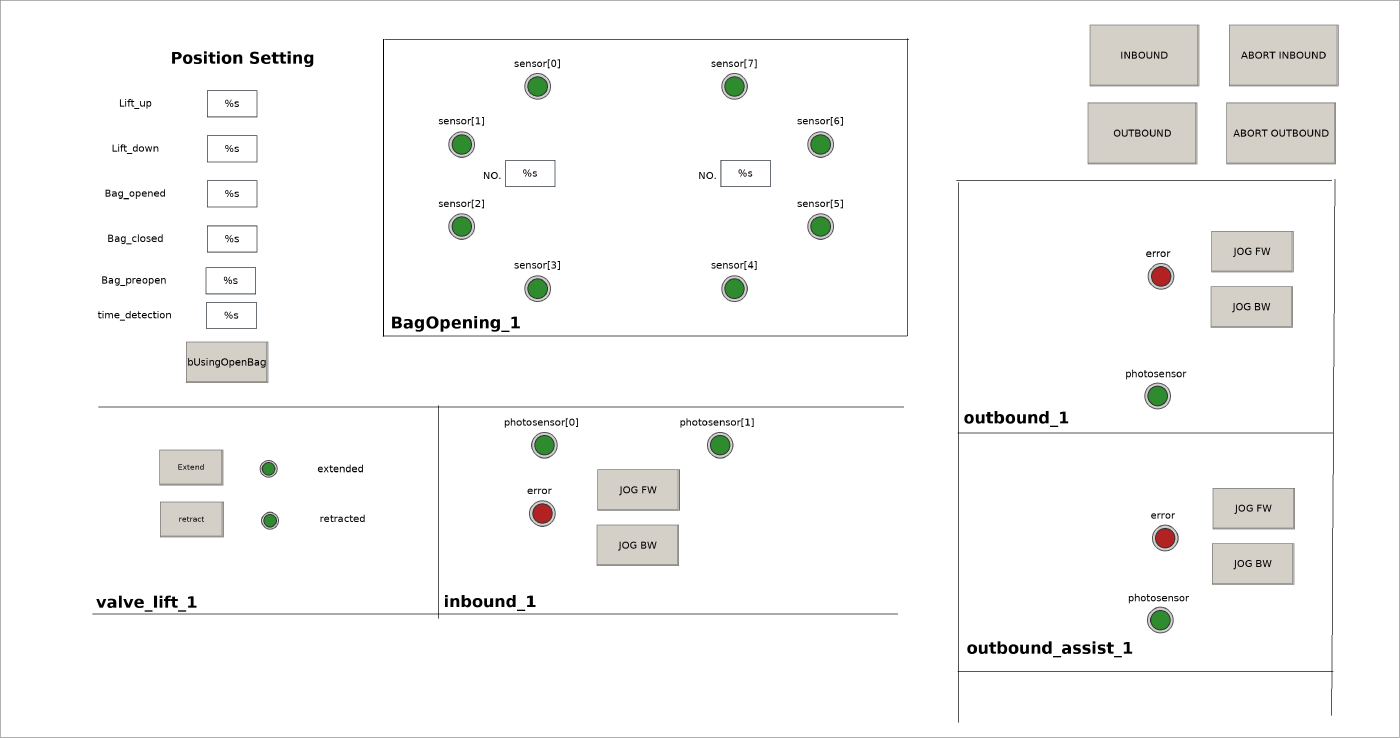
VISUALIZATION v_io_working1  // 2048x1080
    Label (91,855 248x53), "valve_lift_1"
    Button (233,658 93x52), "Extend", colour toggle: GVL.fb_working1.valve_lift.extend
        OnMouseDown: execute { GVL.fb_working1.valve_lift.extend := TRUE; GVL.fb_working1.valve_lift.retract := FALSE; }
    Button (234,734 93x52), "retract", colour toggle: GVL.fb_working1.valve_lift.retract
        OnMouseDown: execute { GVL.fb_working1.valve_lift.extend 	:= FALSE; GVL.fb_working1.valve_lift.retract 	:= TRUE; }
    Lamp1 (378,671 30x30), variable: GVL.fb_working1.valve_lift.extended, style: Lamp-Lamp1-Green
    Lamp1 (380,747 30x30), variable: GVL.fb_working1.valve_lift.retracted, style: Lamp-Lamp1-Green
    Label (432,673 132x26), "extended"
    Label (435,746 132x26), "retracted"
    Lamp1 (771,729 45x45), variable: GVL.fb_working1.roller_inbound.roller.err.Q, style: Lamp-Lamp1-Red
    Label (689,705 200x26), "error"
    Line (144,595) (1322,595)
    Button (874,687 120x60), "JOG FW", colour toggle: GVL.fb_working1.roller_inbound.roller.forward
        OnMouseDown: execute { GVL.fb_working1.roller_inbound.roller.forward	:= TRUE; }
        OnMouseUp: execute { GVL.fb_working1.roller_inbound.roller.forward	:= FALSE; }
    Button (873,768 120x60), "JOG BW", colour toggle: GVL.fb_working1.roller_inbound.roller.backward
        OnMouseDown: execute { GVL.fb_working1.roller_inbound.roller.backward	:= TRUE; }
        OnMouseUp: execute { GVL.fb_working1.roller_inbound.roller.backward	:= FALSE; }
    Lamp1 (774,629 45x45), variable: GVL.fb_working1.roller_inbound.photo_sensor[0].Q, style: Lamp-Lamp1-Green
    Label (692,605 200x26), "photosensor[0]"
    Lamp1 (1031,629 45x45), variable: GVL.fb_working1.roller_inbound.photo_sensor[1].Q, style: Lamp-Lamp1-Green
    Label (949,605 200x26), "photosensor[1]"
    Label (607,855 220x51), "inbound_1"
    Lamp1 (1676,382 45x45), variable: GVL.fb_working1.roller_outbound.roller.err.Q, style: Lamp-Lamp1-Red
    Label (1594,358 200x26), "error"
    Line (1399,264) (1948,264)
    Button (1772,338 120x60), "JOG FW", colour toggle: GVL.fb_working1.roller_outbound.roller.forward
        OnMouseDown: execute { GVL.fb_working1.roller_outbound.roller.forward	:= TRUE; }
        OnMouseUp: execute { GVL.fb_working1.roller_outbound.roller.forward	:= FALSE; }
    Button (1771,419 120x60), "JOG BW", colour toggle: GVL.fb_working1.roller_outbound.roller.backward
        OnMouseDown: execute { GVL.fb_working1.roller_outbound.roller.backward	:= TRUE; }
        OnMouseUp: execute { GVL.fb_working1.roller_outbound.roller.backward	:= FALSE; }
    Lamp1 (1671,557 45x45), variable: GVL.fb_working1.photo_sensor_tote_detection.Q, style: Lamp-Lamp1-Green
    Label (1591,534 200x26), "photosensor"
    Label (1375,587 224x49), "outbound_1"
    Lamp1 (1682,765 45x45), variable: GVL.fb_working1.roller_outbound_assist.roller.err.Q, style: Lamp-Lamp1-Red
    Label (1601,741 200x26), "error"
    Line (1401,633) (1950,633)
    Button (1774,714 120x60), "JOG FW", colour toggle: GVL.fb_working1.roller_outbound_assist.roller.forward
        OnMouseDown: execute { GVL.fb_working1.roller_outbound_assist.roller.forward	:= TRUE; }
        OnMouseUp: execute { GVL.fb_working1.roller_outbound_assist.roller.forward	:= FALSE; }
    Button (1773,795 120x60), "JOG BW", colour toggle: GVL.fb_working1.roller_outbound_assist.roller.backward
        OnMouseDown: execute { GVL.fb_working1.roller_outbound_assist.roller.backward	:= TRUE; }
        OnMouseUp: execute { GVL.fb_working1.roller_outbound_assist.roller.backward	:= FALSE; }
    Line (1401,982) (1950,982)
    Label (1336,940 400x75), "outbound_assist_1"
    Line (641,905) (641,593)
    Line (1948,1047) (1953,262)
    Line (1402,1057) (1402,267)
    Line (135,898) (1313,898)
    Lamp1 (764,400 45x45), variable: GVL.fb_working1.BagOpening_Detection[3], style: Lamp-Lamp1-Green
    Label (686,375 200x26), "sensor[3]"
    Lamp1 (1052,400 45x45), variable: GVL.fb_working1.BagOpening_Detection[4], style: Lamp-Lamp1-Green
    Label (974,375 200x26), "sensor[4]"
    Lamp1 (1178,309 45x45), variable: GVL.fb_working1.BagOpening_Detection[5], style: Lamp-Lamp1-Green
    Label (1100,285 200x26), "sensor[5]"
    Lamp1 (1178,189 45x45), variable: GVL.fb_working1.BagOpening_Detection[6], style: Lamp-Lamp1-Green
    Label (1100,164 200x26), "sensor[6]"
    Lamp1 (1052,104 45x45), variable: GVL.fb_working1.BagOpening_Detection[7], style: Lamp-Lamp1-Green
    Label (974,80 200x26), "sensor[7]"
    Lamp1 (764,104 45x45), variable: GVL.fb_working1.BagOpening_Detection[0], style: Lamp-Lamp1-Green
    Label (686,80 200x26), "sensor[0]"
    Lamp1 (653,189 45x45), variable: GVL.fb_working1.BagOpening_Detection[1], style: Lamp-Lamp1-Green
    Label (575,164 200x26), "sensor[1]"
    Lamp1 (653,309 45x45), variable: GVL.fb_working1.BagOpening_Detection[2], style: Lamp-Lamp1-Green
    Label (575,285 200x26), "sensor[2]"
    Line (562,57) (1329,57)
    Line (561,492) (561,57)
    Line (560,491) (1327,491)
    Line (1328,491) (1328,56)
    Rectangle (303,132 73x39), "%s", text variable: GVL.fb_working1.rPos_lift_up
        OnMouseClick: write the text variable via Default, min GVL.fb_working1.rMin_lift, max GVL.fb_working1.rMax_lift
    Rectangle (303,198 73x39), "%s", text variable: GVL.fb_working1.rPos_lift_down
        OnMouseClick: write the text variable via Default, min GVL.fb_working1.rMin_lift, max GVL.fb_working1.rMax_lift
    Rectangle (303,264 73x39), "%s", text variable: GVL.fb_working1.rPos_bag_opened
        OnMouseClick: write the text variable via Default, min GVL.fb_working1.rMin_bag, max GVL.fb_working1.rMax_bag
    Rectangle (303,330 73x39), "%s", text variable: GVL.fb_working1.rPos_bag_closed
        OnMouseClick: write the text variable via Default, min GVL.fb_working1.rMin_bag, max GVL.fb_working1.rMax_bag
    Label (98,138 200x26), "Lift_up"
    Label (98,204 200x26), "Lift_down"
    Label (98,270 200x26), "Bag_opened"
    Label (98,336 200x26), "Bag_closed"
    Label (180,72 350x26), "Position Setting"
    Rectangle (739,234 73x39), "%s", text variable: GVL.fb_working1.iSensor_detection_setting[0]
        OnMouseClick: write the text variable via Default, min 3, max 4
    Label (670,244 100x26), "NO."
    Rectangle (1054,234 73x39), "%s", text variable: GVL.fb_working1.iSensor_detection_setting[1]
        OnMouseClick: write the text variable via Default, min 3, max 4
    Label (985,244 100x26), "NO."
    Label (454,432 426x81), "BagOpening_1"
    Lamp1 (1675,885 45x45), variable: GVL.fb_working1.roller_outbound.photo_sensor.Q, style: Lamp-Lamp1-Green
    Label (1595,862 200x26), "photosensor"
    Rectangle (301,391 73x39), "%s", text variable: GVL.fb_working1.rPos_bag_preopen
        OnMouseClick: write the text variable via Default, min GVL.fb_working1.rMin_bag, max 15
    Label (96,397 200x26), "Bag_preopen"
    Rectangle (302,442 73x39), "%s", text variable: GVL.fb_working1.iDelay_sensor_detection
        OnMouseClick: write the text variable via Default, min 100, max 500
    Label (97,448 200x26), "time_detection"
    Button (1594,36 160x90), "INBOUND", colour toggle: MAIN.tote_1.bInbound
        OnMouseUp: execute { MAIN.tote_1.bInbound	:= TRUE; }
    Button (1591,150 160x90), "OUTBOUND", colour toggle: MAIN.tote_1.bOutbound
        OnMouseUp: execute { MAIN.tote_1.bOutbound	:= TRUE; }
    Button (1798,36 160x90), "ABORT INBOUND", colour toggle: MAIN.tote_1.bAbortInbound
        OnMouseUp: execute { MAIN.tote_1.bAbortInbound	:= TRUE; }
    Button (1794,150 160x90), "ABORT OUTBOUND", colour toggle: MAIN.tote_1.bAbortOutbound
        OnMouseUp: execute { MAIN.tote_1.bAbortOutbound	:= TRUE; }
    Button (272,500 120x60), "bUsingOpenBag", colour toggle: GVL.fb_working1.bUsingOpenBag
        toggle GVL.fb_working1.bUsingOpenBag
END_VISUALIZATION
